(* IEC 61131-3 sources: Yaha/Documentation/Infomaterial/OSCAT/pcworx_basic_333/module_export (part 3) *)

(* ---- DT_TO_STRF.ST ---- *)
(*@PROPERTIES_EX@
TYPE: POU
LOCALE: 0
IEC_LANGUAGE: ST
PLC_TYPE: independent
PROC_TYPE: independent
GROUP: STRINGS
*)
(*@KEY@:DESCRIPTION*)
version 1.1	19. oct. 2008
programmer 	hugo
tested by	oscat

DT_TO_STRINGF converts a DATETIME input to a formatted string
(*@KEY@:END_DESCRIPTION*)
FUNCTION_BLOCK DT_TO_STRF

(*Group:NewGroup*)

VAR_INPUT
	DTI :	UDINT;
	MS :	INT;
	FMT :	STRING;
	LANG :	INT;
END_VAR

VAR_OUTPUT
	DT_TO_STRF :	STRING;
END_VAR

VAR
	FILL :	oscat_STRING1 := STRING#'0';
	BLANK :	oscat_STRING1 := STRING#' ';
	ly :	INT;
	dx :	UDINT;
	fs :	oscat_STRING10;
	fs_tmp :	oscat_STRING10;
	td :	UDINT;
	tmp :	INT;
	pos :	INT;
	f :	INT;
	CODE :	CODE;
	MONTH_TO_STRING :	MONTH_TO_STRING;
	WEEKDAY_TO_STRING :	WEEKDAY_TO_STRING;
END_VAR

(*@KEY@: WORKSHEET
NAME: DT_TO_STRF
IEC_LANGUAGE: ST
*)
IF LANG < 1 THEN ly := 1; ELSE ly := MIN(2, LANG); END_IF;

(* decode date and time information *)
dx := DT_TO_DATE(DTI);
td := DT_TO_TOD(DTI);

(* parse the format string *)
DT_TO_STRF := FMT;
pos := FIND(DT_TO_STRF, '#');
WHILE pos > 0 DO
	(* retrieve format identifier *)
    CODE(STR:=DT_TO_STRF,POS:=pos + 1);
    f := _BYTE_TO_INT(CODE.CODE);
	(* generate the return string according to the format character *)
	fs := '';
	CASE f OF
         0: RETURN; (* illegal character index *)

		65 : (* letter A retunrs the year in 4 digits *)
			fs := INT_TO_STRING(YEAR_OF_DATE(dx),'%d');
		66 : (* letter B returns the year in exactly 2 digits *)
			fs := RIGHT(INT_TO_STRING(YEAR_OF_DATE(dx),'%02d'),2);
		67 : (* letter C returns the month with 1 or 2 digits *)
			fs := INT_TO_STRING(MONTH_OF_DATE(dx),'%d');
		68 : (* letter D returns the month with exactly 2 digits *)
			fs := INT_TO_STRING(MONTH_OF_DATE(dx),'%02d');
		69 : (* letter E returns the month with 3 characters *)
            MONTH_TO_STRING(MTH:=MONTH_OF_DATE(dx),LANG:=ly,LX:=3);
            fs:=MONTH_TO_STRING.MONTH_TO_STRING;
		70 : (* letter F returns the month with all characters *)
            MONTH_TO_STRING(MTH:=MONTH_OF_DATE(dx),LANG:=ly,LX:=0);
            fs:=MONTH_TO_STRING.MONTH_TO_STRING;
		71 : (* letter G returns the day with up to 2 digits *)
			fs := INT_TO_STRING(DAY_OF_MONTH(dx),'%d');
		72 : (* letter H returns the day of the month with exactly 2 digits *)
			fs := INT_TO_STRING(DAY_OF_MONTH(dx),'%d');
			IF LEN(fs) < 2 THEN fs_tmp:=fs; fs := CONCAT(FILL, fs_tmp); END_IF;
		73 : (* letter I returns the weekday as the number 1..7 1 = monday *)
			fs := INT_TO_STRING(DAY_OF_WEEK(dx),'%d');
		74 : (* letter J returns the weekday in 2 character writing *)
            WEEKDAY_TO_STRING(WDAY:=DAY_OF_WEEK(dx),LANG:=ly,LX:=2);
            fs := WEEKDAY_TO_STRING.WEEKDAY_TO_STRING;
		75 : (* letter K returns the weekday with all characters *)
            WEEKDAY_TO_STRING(WDAY:=DAY_OF_WEEK(dx),LANG:=ly,LX:=0);
            fs := WEEKDAY_TO_STRING.WEEKDAY_TO_STRING;
		76 : (* letter L returns AM or PM for the given DateTime *)
			IF td >= UDINT#43200000 THEN fs := 'PM'; ELSE fs := 'AM'; END_IF;
		77 : (* letter M returns the hour in 1 or 2 digit form 0..24h *)
			fs := INT_TO_STRING(HOUR(td),'%d');
		78 : (* letter N returns the hour in exactly 2 digit form 0..24h *)
			fs := INT_TO_STRING(HOUR(td),'%d');
			IF LEN(fs) < 2 THEN fs_tmp:=fs; fs := CONCAT(FILL, fs_tmp); END_IF;
		79 : (* letter O returns the hour in 1 or 2 digit form 0..12h *)
			tmp := HOUR(td) MOD 12;
			IF tmp = 0 THEN tmp := 12; END_IF;
			fs := INT_TO_STRING(tmp,'%d');
		80 : (* letter P returns the hour in exactly 2 digit form 0..12h *)
			tmp := HOUR(td) MOD 12;
			IF tmp = 0 THEN tmp := 12; END_IF;
			fs := INT_TO_STRING(tmp,'%d');
			IF LEN(fs) < 2 THEN fs_tmp:=fs; fs := CONCAT(FILL, fs_tmp); END_IF;
		81 : (* letter Q returns the minute of the hour in 1 or two digit form *)
			fs := INT_TO_STRING(MINUTE(td),'%d');
		82 : (* letter R returns the minute of the hour in exactly two digit form *)
			fs := INT_TO_STRING(MINUTE(td),'%d');
			IF LEN(fs) < 2 THEN fs_tmp:=fs; fs := CONCAT(FILL, fs_tmp); END_IF;
		83 : (* letter S returns the second of the minute in 1 or two digit form *)
			fs := INT_TO_STRING(REAL_TO_INT(SECOND(td)),'%d');
		84 : (* letter T returns the second of the minute in exactly two digit form *)
			fs := INT_TO_STRING(REAL_TO_INT(SECOND(td)),'%d');
			IF LEN(fs) < 2 THEN fs_tmp:=fs; fs := CONCAT(FILL, fs_tmp); END_IF;
		85 : (* letter U returns the milliseconds in 1 to 3 digits *)
			fs := INT_TO_STRING(MS,'%d');
		86 : (* letter V returns the milliseconds in exactly 3 digit form *)
			fs := INT_TO_STRING(MS,'%03d');
		87 : (* letter W returns the day of the month with exactly 2 digits first digit is filled with blank if necessary *)
			fs := INT_TO_STRING(DAY_OF_MONTH(dx),'%d');
			IF LEN(fs) < 2 THEN fs_tmp:=fs; fs := CONCAT(BLANK, fs_tmp); END_IF;
		88 : (* letter X returns the month with exactly 2 digits first digit is filled with blank if necessary *)
			fs := INT_TO_STRING(MONTH_OF_DATE(dx),'%d');
			IF LEN(fs) < 2 THEN fs_tmp:=fs; fs := CONCAT(BLANK, fs_tmp); END_IF;
	END_CASE;
	DT_TO_STRF := REPLACE(DT_TO_STRF, fs, 2, pos);
	pos := FIND(DT_TO_STRF, '#');
END_WHILE;

(* revision history
hm	7. oct. 2008	rev 1.0
	original version

hm	19. oct. 2008	rev 1.1
	changed language setup constants
*)
(*@KEY@: END_WORKSHEET *)
END_FUNCTION_BLOCK

(* ---- DT_TO_STRING.ST ---- *)
(*@PROPERTIES_EX@
TYPE: POU
LOCALE: 0
IEC_LANGUAGE: ST
PLC_TYPE: independent
PROC_TYPE: independent
GROUP: EMULATION
*)
(*@KEY@:DESCRIPTION*)

(*@KEY@:END_DESCRIPTION*)
FUNCTION_BLOCK DT_TO_STRING

(*Group:Default*)

VAR_INPUT
	IDT :	UDINT;
END_VAR

VAR_OUTPUT
	DT_STRING :	STRING;
END_VAR

VAR
	st_tmp1 :	STRING;
	st_tmp2 :	STRING;
END_VAR

(*@KEY@: WORKSHEET
NAME: DT_TO_STRING
IEC_LANGUAGE: ST
*)
st_tmp2 := CONCAT(INT_TO_STRING(YEAR_OF_DATE(IDT),'%04d-'),INT_TO_STRING(MONTH_OF_DATE(IDT),'%02d-'));
st_tmp1 := CONCAT(INT_TO_STRING(day_of_month(IDT),'%02d-'),INT_TO_STRING(hour_of_DT(IDT),'%02d:'));
st_tmp2 := CONCAT(st_tmp2,st_tmp1);
st_tmp1 := CONCAT(INT_TO_STRING(minute_of_DT(IDT),'%02d:'),INT_TO_STRING(second_of_DT(IDT),'%02d'));
st_tmp2 := CONCAT(st_tmp2,st_tmp1);
DT_STRING := st_tmp2;
(*@KEY@: END_WORKSHEET *)
END_FUNCTION_BLOCK

(* ---- DW_TO_REAL.ST ---- *)
(*@PROPERTIES_EX@
TYPE: POU
LOCALE: 0
IEC_LANGUAGE: ST
PLC_TYPE: independent
PROC_TYPE: independent
GROUP: LOGIC.GATE_LOGIC
*)
(*@KEY@:DESCRIPTION*)
version 1.0	18. apr. 2008
programmer 	hugo
tested by	tobias

this function converts a DWORD to REAL in a bitwise manner.
(*@KEY@:END_DESCRIPTION*)
FUNCTION_BLOCK DW_TO_REAL

(*Group:Default*)

VAR_INPUT
	X :	DWORD;
END_VAR

VAR_OUTPUT
	DW_TO_REAL :	REAL;
END_VAR

VAR
	BUF_TO_REAL :	BUF_TO_REAL;
	i :	INT;
END_VAR

(*@KEY@: WORKSHEET
NAME: DW_TO_REAL
IEC_LANGUAGE: ST
*)
(* BUF_TO_REAL muss mit positiver Flanke gstartet werden darum wird dieser *)
(* einmal mit REQ=0 und dann mit REQ=1 aufgerufen                          *)
(* somit kann in jeden zyklus kopiert werden                               *)

FOR I := 0 TO 1 DO
  BUF_TO_REAL.REQ        := I > 0;
  BUF_TO_REAL.BUF_FORMAT := FALSE;
  BUF_TO_REAL.BUF_OFFS   := DINT#0;
  BUF_TO_REAL.BUF_CNT    := DINT#4;
  BUF_TO_REAL.BUFFER     := X;
  BUF_TO_REAL.DST        := DW_TO_REAL;
  BUF_TO_REAL();
  X           := BUF_TO_REAL.BUFFER;
  DW_TO_REAL  := BUF_TO_REAL.DST;
END_FOR;
(*@KEY@: END_WORKSHEET *)
END_FUNCTION_BLOCK

(* ---- DWORD_TO_STRB.ST ---- *)
(*@PROPERTIES_EX@
TYPE: POU
LOCALE: 0
IEC_LANGUAGE: ST
PLC_TYPE: independent
PROC_TYPE: independent
GROUP: STRINGS
*)
(*@KEY@:DESCRIPTION*)
version 1.3	20. jun. 2008
programmer 	hugo
tested by	oscat

DWORD_TO_STRINGB converts a DWORD to a String of Bits represented by '0' and '1' s.
The lowest order bit will be on the right and the high order bit on the left.
(*@KEY@:END_DESCRIPTION*)
FUNCTION_BLOCK DWORD_TO_STRB

(*Group:Default*)

VAR_INPUT
	IN :	DWORD;
END_VAR

VAR_OUTPUT
	DWORD_TO_STRB :	oscat_STRING32;
END_VAR

VAR
	i :	INT;
END_VAR

(*@KEY@: WORKSHEET
NAME: DWORD_TO_STRB
IEC_LANGUAGE: ST
*)
DWORD_TO_STRB :='';
FOR i := 1 TO 32 DO
    IF (in AND DWORD#16#8000_0000) > DWORD#0 THEN
        DWORD_TO_STRB := CONCAT(DWORD_TO_STRB,'1');
    ELSE
        DWORD_TO_STRB := CONCAT(DWORD_TO_STRB,'0');
    END_IF;
	in := SHL(in, 1);
END_FOR;

(* revision history
hm		9.6.2007	rev 1.0
	original version

hm		15.dec 2007	rev 1.1
	changed code for better performance

hm	29. mar. 2008	rev 1.2
	changed STRING to STRING(32)

hm	20. jun. 2008	rev 1.3
	performance improvement

*)
(*@KEY@: END_WORKSHEET *)
END_FUNCTION_BLOCK

(* ---- DWORD_TO_STRF.ST ---- *)
(*@PROPERTIES_EX@
TYPE: POU
LOCALE: 0
IEC_LANGUAGE: ST
PLC_TYPE: independent
PROC_TYPE: independent
GROUP: STRINGS
*)
(*@KEY@:DESCRIPTION*)
version 1.0	26 jan 2007
programmer 	hugo
tested by		tobias

dword_to_strF converts a DWORD, BYTE or Word to a fixed length String.
the string will be filled with leading zeroes to achieve the fixed length, or if too long, the lowest digits will be used.
the maximum allowed length is 20 mdigits.

for example:	dword_to_strf(123,4) = '0123'
				dword_to_strf(123,2) = '23'
(*@KEY@:END_DESCRIPTION*)
FUNCTION_BLOCK DWORD_TO_STRF

(*Group:Default*)

VAR_INPUT
	IN :	DWORD;
	N :	INT;
END_VAR

VAR_OUTPUT
	DWORD_TO_STRF :	STRING;
END_VAR

VAR
	FIX :	FIX;
END_VAR

(*@KEY@: WORKSHEET
NAME: DWORD_TO_STRF
IEC_LANGUAGE: ST
*)
(* limit N to max 20 characters *)
(* convert dword to string first and cut to length N *)
FIX(str:=DWORD_TO_STRING(in,'%u'),L:=LIMIT(0,N,20),C:=BYTE#48,M:=1);
DWORD_TO_STRF:=FIX.FIX;

(* old code

temp := DWORD_TO_STRING(in,STRING#'%u');
L := LEN(temp);
IF N < L THEN
    temp :=RIGHT(temp,N);
    L := N;
END_IF;

WHILE L < N DO
    temp2 := temp;
	temp := CONCAT('0', temp2);
	L := L + 1;
END_WHILE;
DWORD_TO_STRF := temp;

*)

(* revision history
hm	26. jan.2007	rev 1.0
	original version

hm	29. mar. 2008	rev 1.1
	changed STRING to STRING(20)
	limit the output string to max 20 digits
*)
(*@KEY@: END_WORKSHEET *)
END_FUNCTION_BLOCK

(* ---- DWORD_TO_STRH.ST ---- *)
(*@PROPERTIES_EX@
TYPE: POU
LOCALE: 0
IEC_LANGUAGE: ST
PLC_TYPE: independent
PROC_TYPE: independent
GROUP: STRINGS
*)
(*@KEY@:DESCRIPTION*)
version 1.3	29. mar. 2008
programmer 	hugo
tested by	tobias

DWORD_TO_STRINGH converts a DWORD to a String of Hexadecimal represented by '0' .. '9' and 'A' .. 'F'.
The lowest order Character will be on the right and the high order Character on the left.
(*@KEY@:END_DESCRIPTION*)
FUNCTION_BLOCK DWORD_TO_STRH

(*Group:Default*)

VAR_INPUT
	IN :	DWORD;
END_VAR

VAR_OUTPUT
	DWORD_TO_STRH :	STRING;
END_VAR

(*@KEY@: WORKSHEET
NAME: DWORD_TO_STRH
IEC_LANGUAGE: ST
*)
DWORD_TO_STRH:=DWORD_TO_STRING(IN,'%08X');

(* old code
temp :='';
FOR i := 1 TO 8 DO
	X := DWORD_TO_INT(in AND DWORD#2#1111);
	IF X <= 9 THEN X := X + 48; ELSE X := X + 55; END_IF;

    CHR(C:=INT_TO_BYTE(X));

    temp2 := temp;
	temp := CONCAT(CHR.CHR, temp2);
	in := SHR(in,4);
END_FOR;
DWORD_TO_STRH := temp;
*)

(* revision history
hm	9. jun. 2007	rev 1.0
	original version

hm	11. sep. 2007	rev 1.1
	changed coding for compatibility with twincat, concat cannot support a function as an argument.

hm	15. dec. 2007	rev 1.2
	changed code for better performance

hm	29. mar. 2008	rev 1.3
	changed STRING to STRING(8)

*)
(*@KEY@: END_WORKSHEET *)
END_FUNCTION_BLOCK

(* ---- ENERGY.ST ---- *)
(*@PROPERTIES_EX@
TYPE: POU
LOCALE: 0
IEC_LANGUAGE: ST
PLC_TYPE: independent
PROC_TYPE: independent
GROUP: ENGINEERING.CONVERSION
*)
(*@KEY@:DESCRIPTION*)
version 1.2	16. jan. 2010
programmer 	hugo
tested by	oscat

this function converts different energy units
any unused input can simply be left open.
different inputs connected at the same time will be added up.
(*@KEY@:END_DESCRIPTION*)
FUNCTION_BLOCK ENERGY

(*Group:Default*)

VAR_INPUT
	J :	REAL;
	C :	REAL;
	WH :	REAL;
END_VAR

VAR_OUTPUT
	YJ :	REAL;
	YC :	REAL;
	YWH :	REAL;
END_VAR

(*@KEY@: WORKSHEET
NAME: ENERGY
IEC_LANGUAGE: ST
*)
YJ := J + Wh * 3600.0 + C * 4.1868;
YC := YJ * 0.238845896627496;
YWh := YJ * 2.7777777778E-004;

(*
Arbeit, Energie, Joule* J 1 J = 1 N · m = 1 W · s = (1/3,6) E–6 kW · h = 1 kg · m2/s2
Wärmemenge Kilowattstunde kW · h 1 kW · h = 3,6 MJ = 860 kcal
Elektronvolt eV 1 eV = 160,218 92 E–21 J
Erg erg 1 erg = 1E–7 J
Kalorie calorie 1 calalorie = 4,1868 J = 1,163 E–3 W · h
Therm therm 1 therm = 105,50 · 106 J
*)

(* revision history

hm	27. mar. 2007	rev 1.0
	original version

hm	11. mar. 2009	rev 1.1
	improved code

hm 16. jan 2010	rev 1.2
	avoid the string cal in comments for codesys import bug

*)
(*@KEY@: END_WORKSHEET *)
END_FUNCTION_BLOCK

(* ---- ESR_COLLECT.ST ---- *)
(*@PROPERTIES_EX@
TYPE: POU
LOCALE: 0
IEC_LANGUAGE: ST
PLC_TYPE: independent
PROC_TYPE: independent
GROUP: OTHER
*)
(*@KEY@:DESCRIPTION*)
version 1.4	1. dec. 2009
programmer 	hugo
tested by	tobias

ESR_collect collects esr data from up to 8 esr_mon modules and stroes them in an output array.
the output pos will display the position of the last element in the array. if the array is empty, pos = -1
when to buffer is read by followon modules. pos has to be reset to -1
if the array will be full, the buffer will be refilled starting at position 0.

(*@KEY@:END_DESCRIPTION*)
FUNCTION_BLOCK ESR_COLLECT

(*Group:Default*)

VAR_INPUT
	ESR_0 :	oscat_ESR_3;
	ESR_1 :	oscat_ESR_3;
	ESR_2 :	oscat_ESR_3;
	ESR_3 :	oscat_ESR_3;
	ESR_4 :	oscat_ESR_3;
	ESR_5 :	oscat_ESR_3;
	ESR_6 :	oscat_ESR_3;
	ESR_7 :	oscat_ESR_3;
	RST :	BOOL;
END_VAR

VAR_IN_OUT
	POS :	INT;
END_VAR

VAR_OUTPUT
	ESR_OUT :	oscat_ESR_31;
END_VAR

VAR
	cnt :	INT := -1;
	max_in :	INT := 3;
	max_out :	INT := 32;
END_VAR

(*@KEY@: WORKSHEET
NAME: ESR_COLLECT
IEC_LANGUAGE: ST
*)
IF rst OR cnt < 0 THEN
	pos := -1;
ELSE
	FOR cnt := 0 TO max_in DO
	IF esr_0[cnt].typ > BYTE#0 THEN pos := INC1(pos, max_out); esr_out[pos] := esr_0[cnt]; END_IF;
	IF esr_1[cnt].typ > BYTE#0 THEN pos := INC1(pos, max_out); esr_out[pos] := esr_1[cnt]; END_IF;
	IF esr_2[cnt].typ > BYTE#0 THEN pos := INC1(pos, max_out); esr_out[pos] := esr_2[cnt]; END_IF;
	IF esr_3[cnt].typ > BYTE#0 THEN pos := INC1(pos, max_out); esr_out[pos] := esr_3[cnt]; END_IF;
	IF esr_4[cnt].typ > BYTE#0 THEN pos := INC1(pos, max_out); esr_out[pos] := esr_4[cnt]; END_IF;
	IF esr_5[cnt].typ > BYTE#0 THEN pos := INC1(pos, max_out); esr_out[pos] := esr_5[cnt]; END_IF;
	IF esr_6[cnt].typ > BYTE#0 THEN pos := INC1(pos, max_out); esr_out[pos] := esr_6[cnt]; END_IF;
	IF esr_7[cnt].typ > BYTE#0 THEN pos := INC1(pos, max_out); esr_out[pos] := esr_7[cnt]; END_IF;
   END_FOR;
END_IF;

(* revision history
hm	26.jan 2007	rev 1.0
	original version

hm	8. dec 2007	rev 1.1
	added reset input

ks	27. oct. 2008	rev 1.2
	optimized code for performance

ks	12. nov. 2009	rev 1.3
	output pos was not pointing to last value

hm	1. dec. 2009	rev 1.4
	changed pos to be I/O
	reduced output array size to 32 elements
*)
(*@KEY@: END_WORKSHEET *)
END_FUNCTION_BLOCK

(* ---- ESR_MON_B8.ST ---- *)
(*@PROPERTIES_EX@
TYPE: POU
LOCALE: 0
IEC_LANGUAGE: ST
PLC_TYPE: independent
PROC_TYPE: independent
GROUP: OTHER
*)
(*@KEY@:DESCRIPTION*)
version 1.3	1. dec. 2009
programmer 	hugo
tested by	tobias

ESR_mon_B8 monitores up to 8 binary inputs and reports changes with time stamd and adress label.
the module checks 8 inputs for a change and reports all changes with time and adress stamp to the output.
4 events maximum can be collected at once within the same cycle

(*@KEY@:END_DESCRIPTION*)
FUNCTION_BLOCK ESR_MON_B8

(*Group:Default*)

VAR_INPUT
	S0 :	BOOL;
	A0 :	oscat_STRING10;
	S1 :	BOOL;
	A1 :	oscat_STRING10;
	S2 :	BOOL;
	A2 :	oscat_STRING10;
	S3 :	BOOL;
	A3 :	oscat_STRING10;
	S4 :	BOOL;
	A4 :	oscat_STRING10;
	S5 :	BOOL;
	A5 :	oscat_STRING10;
	S6 :	BOOL;
	A6 :	oscat_STRING10;
	S7 :	BOOL;
	A7 :	oscat_STRING10;
	DT_IN :	UDINT;
END_VAR

VAR_IN_OUT
	ESR_Out :	oscat_ESR_3;
END_VAR

VAR_OUTPUT
	ESR_FLAG :	BOOL;
END_VAR

VAR
	x0 :	BOOL;
	x1 :	BOOL;
	x2 :	BOOL;
	x3 :	BOOL;
	x4 :	BOOL;
	x5 :	BOOL;
	x6 :	BOOL;
	x7 :	BOOL;
	tx :	TIME;
	cnt :	INT;
	T_PLC_MS :	T_PLC_MS;
END_VAR

(*@KEY@: WORKSHEET
NAME: ESR_MON_B8
IEC_LANGUAGE: ST
*)
(* read system timer *)
T_PLC_MS();
tx:= UDINT_TO_TIME(T_PLC_MS.T_PLC_MS);

ESR_Flag := FALSE;
esr_out[3].typ := BYTE#0;
esr_out[2].typ := BYTE#0;
esr_out[1].typ := BYTE#0;
esr_out[0].typ := BYTE#0;
cnt := 0;

(* check if inputs have chaged and fill buffer *)
IF s0 <> X0 THEN
	esr_out[cnt].typ := INT_TO_BYTE(10 + BOOL_TO_INT(s0));
	esr_out[cnt].adress := a0;
	esr_out[cnt].DS := DT_in;
	esr_out[cnt].TS := TX;
	X0 := S0;
	cnt := cnt + 1;
	esr_flag := TRUE;
END_IF;
IF s1 <> X1 THEN
	esr_out[cnt].typ := INT_TO_BYTE(10 + BOOL_TO_INT(s1));
	esr_out[cnt].adress := a1;
	esr_out[cnt].DS := DT_in;
	esr_out[cnt].TS := TX;
	X1 := S1;
	cnt := cnt + 1;
	esr_flag := TRUE;
END_IF;
IF s2 <> X2 THEN
	esr_out[cnt].typ := INT_TO_BYTE(10 + BOOL_TO_INT(s2));
	esr_out[cnt].adress := a2;
	esr_out[cnt].DS := DT_in;
	esr_out[cnt].TS := TX;
	X2 := S2;
	cnt := cnt + 1;
	esr_flag := TRUE;
END_IF;
IF s3 <> X3 THEN
	esr_out[cnt].typ := INT_TO_BYTE(10 + BOOL_TO_INT(s3));
	esr_out[cnt].adress := a3;
	esr_out[cnt].DS := DT_in;
	esr_out[cnt].TS := TX;
	X3 := S3;
	cnt := cnt + 1;
	esr_flag := TRUE;
END_IF;
IF s4 <> X4 AND cnt < 4 THEN
	esr_out[cnt].typ := INT_TO_BYTE(10 + BOOL_TO_INT(s4));
	esr_out[cnt].adress := a4;
	esr_out[cnt].DS := DT_in;
	esr_out[cnt].TS := TX;
	X4 := S4;
	cnt := cnt + 1;
	esr_flag := TRUE;
END_IF;
IF s5 <> X5  AND cnt < 4 THEN
	esr_out[cnt].typ := INT_TO_BYTE(10 + BOOL_TO_INT(s5));
	esr_out[cnt].adress := a5;
	esr_out[cnt].DS := DT_in;
	esr_out[cnt].TS := TX;
	X5 := S5;
	cnt := cnt + 1;
	esr_flag := TRUE;
END_IF;
IF s6 <> X6  AND cnt < 4 THEN
	esr_out[cnt].typ := INT_TO_BYTE(10 + BOOL_TO_INT(s6));
	esr_out[cnt].adress := a6;
	esr_out[cnt].DS := DT_in;
	esr_out[cnt].TS := TX;
	X6 := S6;
	cnt := cnt + 1;
	esr_flag := TRUE;
END_IF;
IF s7 <> X7  AND cnt < 4 THEN
	esr_out[cnt].typ := INT_TO_BYTE(10 + BOOL_TO_INT(s7));
	esr_out[cnt].adress := a7;
	esr_out[cnt].DS := DT_in;
	esr_out[cnt].TS := TX;
	X7 := S7;
	cnt := cnt + 1;
	esr_flag := TRUE;
END_IF;

(* revision history
hm	26. jan 2007	rev 1.0
	original version

hm	17. sep 2007	rev 1.1
	replaced time() with T_PLC_MS() for compatibility reasons

hm	22. oct. 2008	rev 1.2
	optimized code

hm	1.dec. 2009	rev 1.3
	changed esr_out to be I/O

*)
(*@KEY@: END_WORKSHEET *)
END_FUNCTION_BLOCK

(* ---- ESR_MON_R4.ST ---- *)
(*@PROPERTIES_EX@
TYPE: POU
LOCALE: 0
IEC_LANGUAGE: ST
PLC_TYPE: independent
PROC_TYPE: independent
GROUP: OTHER
*)
(*@KEY@:DESCRIPTION*)
version 1.4	1. dec. 2009
programmer 	hugo
tested by	tobias

ESR_mon_R4 monitores up to 4 Real inputs and reports changes with time stamd and adress label.
the module checks 4 inputs for a change of more than the specified sensitivity S and reports all changes with time and adress stamp to the output.

(*@KEY@:END_DESCRIPTION*)
FUNCTION_BLOCK ESR_MON_R4

(*Group:Default*)

VAR_INPUT
	R0 :	REAL;
	A0 :	oscat_STRING10;
	S0 :	REAL;
	R1 :	REAL;
	A1 :	oscat_STRING10;
	S1 :	REAL;
	R2 :	REAL;
	A2 :	oscat_STRING10;
	S2 :	REAL;
	R3 :	REAL;
	A3 :	oscat_STRING10;
	S3 :	REAL;
	DT_IN :	UDINT;
END_VAR

VAR_IN_OUT
	ESR_OUT :	oscat_ESR_3;
END_VAR

VAR_OUTPUT
	ESR_FLAG :	BOOL;
END_VAR

VAR
	x0 :	REAL;
	x1 :	REAL;
	x2 :	REAL;
	x3 :	REAL;
	tx :	TIME;
	cnt :	INT;
	T_PLC_MS :	T_PLC_MS;
	REAL_TO_DW :	REAL_TO_DW;
	tmp :	DWORD;
END_VAR

(*@KEY@: WORKSHEET
NAME: ESR_MON_R4
IEC_LANGUAGE: ST
*)
T_PLC_MS();
tx:= UDINT_TO_TIME(T_PLC_MS.T_PLC_MS);

ESR_Flag := FALSE;
esr_out[3].typ := BYTE#0;
esr_out[2].typ := BYTE#0;
esr_out[1].typ := BYTE#0;
esr_out[0].typ := BYTE#0;
cnt := 0;

(* check if inputs have chaged and fill buffer *)
IF differ(R0, X0, S0) THEN
    REAL_TO_DW(X:=R0);
    tmp := REAL_TO_DW.REAL_TO_DW;

	esr_out[cnt].typ := BYTE#20;
	esr_out[cnt].adress := a0;
	esr_out[cnt].DS := DT_in;
	esr_out[cnt].TS := TX;
	esr_out[cnt].data[0] := Byte_of_Dword(tmp,BYTE#0);
	esr_out[cnt].data[1] := Byte_of_Dword(tmp,BYTE#1);
	esr_out[cnt].data[2] := Byte_of_Dword(tmp,BYTE#2);
	esr_out[cnt].data[3] := Byte_of_Dword(tmp,BYTE#3);
	X0 := R0;
	cnt := cnt + 1;
	esr_flag := TRUE;
END_IF;
IF differ(R1, X1, S1) THEN
    REAL_TO_DW(X:=R1);
    tmp := REAL_TO_DW.REAL_TO_DW;

	esr_out[cnt].typ := BYTE#20;
	esr_out[cnt].adress := a1;
	esr_out[cnt].DS := DT_in;
	esr_out[cnt].TS := TX;
	esr_out[cnt].data[0] := Byte_of_Dword(tmp,BYTE#0);
	esr_out[cnt].data[1] := Byte_of_Dword(tmp,BYTE#1);
	esr_out[cnt].data[2] := Byte_of_Dword(tmp,BYTE#2);
	esr_out[cnt].data[3] := Byte_of_Dword(tmp,BYTE#3);
	X1 := R1;
	cnt := cnt + 1;
	esr_flag := TRUE;
END_IF;
IF differ(R2, X2, S2) THEN
    REAL_TO_DW(X:=R2);
    tmp := REAL_TO_DW.REAL_TO_DW;

	esr_out[cnt].typ := BYTE#20;
	esr_out[cnt].adress := a2;
	esr_out[cnt].DS := DT_in;
	esr_out[cnt].TS := TX;
	esr_out[cnt].data[0] := Byte_of_Dword(tmp,BYTE#0);
	esr_out[cnt].data[1] := Byte_of_Dword(tmp,BYTE#1);
	esr_out[cnt].data[2] := Byte_of_Dword(tmp,BYTE#2);
	esr_out[cnt].data[3] := Byte_of_Dword(tmp,BYTE#3);
	X2 := R2;
	cnt := cnt + 1;
	esr_flag := TRUE;
END_IF;
IF differ(R3, X3, S3) THEN
    REAL_TO_DW(X:=R2);
    tmp := REAL_TO_DW.REAL_TO_DW;

	esr_out[cnt].typ := BYTE#20;
	esr_out[cnt].adress := a3;
	esr_out[cnt].DS := DT_in;
	esr_out[cnt].TS := TX;
	esr_out[cnt].data[0] := Byte_of_Dword(tmp,BYTE#0);
	esr_out[cnt].data[1] := Byte_of_Dword(tmp,BYTE#1);
	esr_out[cnt].data[2] := Byte_of_Dword(tmp,BYTE#2);
	esr_out[cnt].data[3] := Byte_of_Dword(tmp,BYTE#3);
	X3 := R3;
	cnt := cnt + 1;
	esr_flag := TRUE;
END_IF;

(* revision history
hm	26. jan 2007	rev 1.0
	original version

hm	17. sep. 2007		rev 1.1
	replaced time() with T_PLC_MS() for compatibility reasons

hm	8. dec. 2007		rev 1.2
	corrected an error while esr typ would not be set

hm	16. mar. 2008		rev 1.3
	deleted wrong conversion real_to_dword

hm	1. dec 2009		rev 1.4
	changed esr_out to be I/O

*)

(*@KEY@: END_WORKSHEET *)
END_FUNCTION_BLOCK

(* ---- ESR_MON_X8.ST ---- *)
(*@PROPERTIES_EX@
TYPE: POU
LOCALE: 0
IEC_LANGUAGE: ST
PLC_TYPE: independent
PROC_TYPE: independent
GROUP: OTHER
*)
(*@KEY@:DESCRIPTION*)
version 1.2	1. dec. 2009
programmer 	hugo
tested by	tobias

ESR_MON_X8 is a status and error collector.
the module checks 8 status inputs for a change and reports up to 4 input changes with time and adress stamp to the output.
the mode can be
1 for error only
2 for error and status
3 for error, status and debug
the adress label of the 8 inputs can be configured individually.
(*@KEY@:END_DESCRIPTION*)
FUNCTION_BLOCK ESR_MON_X8

(*Group:Default*)

VAR_INPUT
	S0 :	BYTE;
	A0 :	oscat_STRING10;
	S1 :	BYTE;
	A1 :	oscat_STRING10;
	S2 :	BYTE;
	A2 :	oscat_STRING10;
	S3 :	BYTE;
	A3 :	oscat_STRING10;
	S4 :	BYTE;
	A4 :	oscat_STRING10;
	S5 :	BYTE;
	A5 :	oscat_STRING10;
	S6 :	BYTE;
	A6 :	oscat_STRING10;
	S7 :	BYTE;
	A7 :	oscat_STRING10;
	DT_IN :	UDINT;
	MODE :	BYTE := BYTE#3;
END_VAR

VAR_IN_OUT
	ESR_OUT :	oscat_ESR_3;
END_VAR

VAR_OUTPUT
	ESR_FLAG :	BOOL;
END_VAR

VAR
	x0 :	BYTE;
	x1 :	BYTE;
	x2 :	BYTE;
	x3 :	BYTE;
	x4 :	BYTE;
	x5 :	BYTE;
	x6 :	BYTE;
	x7 :	BYTE;
	tx :	TIME;
	cnt :	INT;
	status_to_ESR :	status_to_ESR;
	T_PLC_MS :	T_PLC_MS;
END_VAR

(*@KEY@: WORKSHEET
NAME: ESR_MON_X8
IEC_LANGUAGE: ST
*)
(* read system timer *)
T_PLC_MS();
tx:= UDINT_TO_TIME(T_PLC_MS.T_PLC_MS);

ESR_Flag := FALSE;
esr_out[3].typ := BYTE#0;
esr_out[2].typ := BYTE#0;
esr_out[1].typ := BYTE#0;
esr_out[0].typ := BYTE#0;
cnt := 0;

(* check if inputs have chaged and fill buffer *)
IF s0 <> X0 AND ((s0 < BYTE#100) OR (S0 > BYTE#99 AND S0 < BYTE#200 AND mode >= BYTE#2) OR (S0 > BYTE#199 AND mode = BYTE#3)) THEN

    status_to_ESR.status := s0;
    status_to_ESR.adress := a0;
    status_to_ESR.DT_in  := DT_in;
    status_to_ESR.TS     := tx;
    status_to_ESR();
    esr_out[cnt] := status_to_ESR.status_to_ESR;

	X0 := S0;
	cnt := cnt + 1;
	esr_flag := TRUE;
END_IF;
IF s1 <> X1 AND ((s1 < BYTE#100) OR (S1 > BYTE#99 AND S1 < BYTE#200 AND mode >= BYTE#2) OR (S1 > BYTE#199 AND mode = BYTE#3)) THEN

    status_to_ESR.status := s1;
    status_to_ESR.adress := a1;
    status_to_ESR.DT_in  := DT_in;
    status_to_ESR.TS     := tx;
    status_to_ESR();
    esr_out[cnt] := status_to_ESR.status_to_ESR;

	X1 := S1;
	cnt := cnt + 1;
	esr_flag := TRUE;
END_IF;
IF s2 <> X2 AND ((s2 < BYTE#100) OR (S2 > BYTE#99 AND S2 < BYTE#200 AND mode >= BYTE#2) OR (S2 > BYTE#199 AND mode = BYTE#3)) THEN

    status_to_ESR.status := s2;
    status_to_ESR.adress := a2;
    status_to_ESR.DT_in  := DT_in;
    status_to_ESR.TS     := tx;
    status_to_ESR();
    esr_out[cnt] := status_to_ESR.status_to_ESR;

	X2 := S2;
	cnt := cnt + 1;
	esr_flag := TRUE;
END_IF;
IF s3 <> X3 AND ((s3 < BYTE#100) OR (S3 > BYTE#99 AND S3 < BYTE#200 AND mode >= BYTE#2) OR (S3 > BYTE#199 AND mode = BYTE#3)) THEN

    status_to_ESR.status := s3;
    status_to_ESR.adress := a3;
    status_to_ESR.DT_in  := DT_in;
    status_to_ESR.TS     := tx;
    status_to_ESR();
    esr_out[cnt] := status_to_ESR.status_to_ESR;

	X3 := S3;
	cnt := cnt + 1;
	esr_flag := TRUE;
END_IF;
IF cnt < 4 AND s4 <> X4 AND ((s4 < BYTE#100) OR (S4 > BYTE#99 AND S4 < BYTE#200 AND mode >= BYTE#2) OR (S4 > BYTE#199 AND mode = BYTE#3)) THEN

    status_to_ESR.status := s4;
    status_to_ESR.adress := a4;
    status_to_ESR.DT_in  := DT_in;
    status_to_ESR.TS     := tx;
    status_to_ESR();
    esr_out[cnt] := status_to_ESR.status_to_ESR;

	X4 := S4;
	cnt := cnt + 1;
	esr_flag := TRUE;
END_IF;
IF cnt < 4 AND s5 <> X5 AND ((s5 < BYTE#100) OR (S5 > BYTE#99 AND S5 < BYTE#200 AND mode >= BYTE#2) OR (S5 > BYTE#199 AND mode = BYTE#3)) THEN

    status_to_ESR.status := s5;
    status_to_ESR.adress := a5;
    status_to_ESR.DT_in  := DT_in;
    status_to_ESR.TS     := tx;
    status_to_ESR();
    esr_out[cnt] := status_to_ESR.status_to_ESR;

	X5 := S5;
	cnt := cnt + 1;
	esr_flag := TRUE;
END_IF;
IF cnt < 4 AND s6 <> X6 AND ((s6 < BYTE#100) OR (S6 > BYTE#99 AND S6 < BYTE#200 AND mode >= BYTE#2) OR (S6 > BYTE#199 AND mode = BYTE#3)) THEN

    status_to_ESR.status := s6;
    status_to_ESR.adress := a6;
    status_to_ESR.DT_in  := DT_in;
    status_to_ESR.TS     := tx;
    status_to_ESR();
    esr_out[cnt] := status_to_ESR.status_to_ESR;

	X6 := S6;
	cnt := cnt + 1;
	esr_flag := TRUE;
END_IF;
IF cnt < 4 AND s7 <> X7 AND ((s7 < BYTE#100) OR (S7 > BYTE#99 AND S7 < BYTE#200 AND mode >= BYTE#2) OR (S7 > BYTE#199 AND mode = BYTE#3)) THEN

    status_to_ESR.status := s7;
    status_to_ESR.adress := a7;
    status_to_ESR.DT_in  := DT_in;
    status_to_ESR.TS     := tx;
    status_to_ESR();
    esr_out[cnt] := status_to_ESR.status_to_ESR;

	X7 := S7;
	cnt := cnt + 1;
	esr_flag := TRUE;
END_IF;

(* revision history
hm	26. jan 2007		rev 1.0
	original version

hm	17. sep 2007	rev 1.1
	replaced time() with T_PLC_MS() for compatibility reasons

hm	1. dec. 2009	rev 1.2
	changed esr_out to be I/O

*)
(*@KEY@: END_WORKSHEET *)
END_FUNCTION_BLOCK

(* ---- EVENTS.ST ---- *)
(*@PROPERTIES_EX@
TYPE: POU
LOCALE: 0
IEC_LANGUAGE: ST
PLC_TYPE: independent
PROC_TYPE: independent
GROUP: TIME_DATE
*)
(*@KEY@:DESCRIPTION*)
version 1.0	18. jan. 2010
programmer 	hugo
tested by	tobias

event checks an array with a list of events and displays the event if today is one.

(*@KEY@:END_DESCRIPTION*)
FUNCTION_BLOCK EVENTS

(*Group:Default*)

VAR_INPUT
	DATE_IN :	UDINT;
	ENA :	BOOL;
END_VAR

VAR_OUTPUT
	Y :	BOOL;
	NAME :	oscat_STRING30;
END_VAR

VAR_IN_OUT
	ELIST :	oscat_HOLIDAY_DATA_0_49;
END_VAR

VAR
	i :	INT;
	last_active :	UDINT;
	size :	INT := 49;
	day_in :	DINT;
	cyr :	INT;
	lday :	DINT;
	check :	oscat_HOLIDAY_DATA;
	y_int :	BOOL;
	name_int :	oscat_STRING30;
END_VAR

(*@KEY@: WORKSHEET
NAME: EVENTS
IEC_LANGUAGE: ST
*)
(* for performance reasons only activate once a day *)
IF last_active <> date_in THEN
	last_active := DATE_IN;
	Y_int := FALSE;
	name_int := '';
	day_in := DAY_OF_DATE(DATE_IN);
	cyr := YEAR_OF_DATE(DATE_IN);

	(* search list for events *)
	FOR i := 0 TO size DO
		check := elist[i];
		lday := DAY_OF_DATE(SET_DATE(cyr,SINT_TO_INT(check.month), SINT_TO_INT(check.day)));
		IF day_in >= lday AND day_in <= lday + SINT_TO_DINT(check.use) - DINT#1 THEN
			y_int := TRUE;
			name_int := check.name;
			EXIT;
		END_IF;
	END_FOR;
END_IF;

IF ENA THEN
	Y := y_int;
	NAME := name_int;
ELSE
	Y := FALSE;
	NAME := '';
END_IF;

(* revision history
hm  18. jan. 2011	rev 1.0
	new module

*)

(*@KEY@: END_WORKSHEET *)
END_FUNCTION_BLOCK

(* ---- EXEC.ST ---- *)
(*@PROPERTIES_EX@
TYPE: POU
LOCALE: 0
IEC_LANGUAGE: ST
PLC_TYPE: independent
PROC_TYPE: independent
GROUP: STRINGS
*)
(*@KEY@:DESCRIPTION*)
version 1.4	29. mar. 2008
programmer 	hugo
tested by	tobias

exec executes a mathematical term and returns the result as a string
the term can only be a simple term without brackets and only one operator
allowed operastors are: (+, -, *, /, ^, sqrt, sin, cos, tan).
(*@KEY@:END_DESCRIPTION*)
FUNCTION_BLOCK EXEC

(*Group:Default*)

VAR_INPUT
	STR :	STRING;
END_VAR

VAR_OUTPUT
	EXEC :	STRING;
END_VAR

VAR
	pos :	INT;
	R1 :	REAL;
	R2 :	REAL;
	operator :	STRING;
	temp :	STRING;
	uppercase :	uppercase;
	trim :	trim;
	findB_num :	findB_num;
	findB_nonum :	findB_nonum;
END_VAR

(*@KEY@: WORKSHEET
NAME: EXEC
IEC_LANGUAGE: ST
*)
(* extract both numbers and operator *)

trim(str:=str);
temp:=trim.trim;

uppercase(str:=temp);
exec:=uppercase.uppercase;

findB_nonum(str:=exec);
pos :=findB_nonum.findB_nonum;

IF pos > 1 THEN
 temp := LEFT(EXEC,pos-1);
 findB_num(str:=temp);
 IF findB_num.findB_num > 0 THEN
   R1 := STRING_TO_REAL(temp);
 END_IF;
END_IF;
temp := RIGHT(exec,LEN(exec)-pos);
R2 := STRING_TO_REAL(temp);
exec := LEFT(exec,pos);

findB_num(str:=exec);
pos :=findB_num.findB_num;
operator := RIGHT(exec,LEN(exec) - pos);
IF EQ_STRING(operator,'') AND LEN(str) = 0 THEN
	exec := '';
	RETURN;
ELSIF EQ_STRING(operator,'') THEN
	exec := str;
	RETURN;
END_IF;
IF EQ_STRING(operator,'^') THEN
	exec := REAL_TO_STRING(EXPT(R1, R2),'%f');
ELSIF EQ_STRING(operator,'SQRT') THEN
	exec := REAL_TO_STRING(SQRT(R2),'%f');
ELSIF EQ_STRING(operator,'SIN') THEN
	exec := REAL_TO_STRING(SIN(r2),'%f');
ELSIF EQ_STRING(operator,'COS') THEN
	exec := REAL_TO_STRING(COS(r2),'%f');
ELSIF EQ_STRING(operator,'TAN') THEN
	exec := REAL_TO_STRING(TAN(R2),'%f');
ELSIF EQ_STRING(operator,'*') THEN
	exec := REAL_TO_STRING(R1 * R2,'%f');
ELSIF EQ_STRING(operator,'/') THEN
	IF R2 <> 0.0 THEN exec := REAL_TO_STRING(R1 / R2,'%f'); ELSE exec := 'ERROR'; END_IF;
ELSIF EQ_STRING(operator,'+') THEN
	exec := REAL_TO_STRING(r1 + r2,'%f');
ELSIF EQ_STRING(operator,'-') THEN
	exec := REAL_TO_STRING(r1 - r2,'%f');
ELSE
	exec := 'ERROR';
END_IF;
IF EQ_STRING(EXEC,'ERROR') THEN
	RETURN;
(* some systems deliver integer instead of real *)
ELSIF FIND(EXEC,'.') = 0 THEN
	EXEC := CONCAT(EXEC, '.0');
(* some systems deliver n. instead of n.0 ! *)
ELSE
 temp := RIGHT(EXEC,1);
 IF EQ_STRING(temp,'.') THEN
    EXEC := CONCAT(EXEC,'0');
  END_IF;
END_IF;

(* revision history

hm 	6.feb 2007		rev 1.1
	cos has to be written in uppercase
	divide by 0 will return an error

hm	5. mar. 2008	rev 1.2
	add a 0 to the string if a '.' is at the end of the string

hm	20. mar. 2008	rev 1.3
	make sure the function always returns a real value in the form of x.y

hm	29. mar. 2008	rev 1.4
	changed STRING to STRING(STRING_LENGTH)
*)
(*@KEY@: END_WORKSHEET *)
END_FUNCTION_BLOCK

(* ---- F_POLY.ST ---- *)
(*@PROPERTIES_EX@
TYPE: POU
LOCALE: 0
IEC_LANGUAGE: ST
PLC_TYPE: independent
PROC_TYPE: independent
GROUP: MATHEMATICAL.FUNCTIONS
*)
(*@KEY@:DESCRIPTION*)
version 1.1	18. mar. 2011
programmer 	hugo
tested by	tobias

this function calculates the polynom C[0] + C[1]*X^1 + C[2]*X^2 * C[3]*X^3 + C[4]*X^4 + C[5]*X^5 + C[6]*X^6 + C[7]*X^7

(*@KEY@:END_DESCRIPTION*)
FUNCTION_BLOCK F_POLY

(*Group:Default*)

VAR_INPUT
	X :	REAL;
	C :	oscat_arr_0_7;
END_VAR

VAR_OUTPUT
	F_POLY :	REAL;
END_VAR

(*@KEY@: WORKSHEET
NAME: F_POLY
IEC_LANGUAGE: ST
*)
F_POLY := ((((((( c[7] * x + c[6] ) * x + c[5] ) * x + c[4] ) * x + c[3] ) * x + c[2] ) * x + c[1] ) * x + c[0] ) ;

(* revision history
hm		20. may. 2008		rev 1.0
	original version

hm	18. mar. 2011	rev 1.1
	improved performance
*)

(*@KEY@: END_WORKSHEET *)
END_FUNCTION_BLOCK

(* ---- FADE.ST ---- *)
(*@PROPERTIES_EX@
TYPE: POU
LOCALE: 0
IEC_LANGUAGE: ST
PLC_TYPE: independent
PROC_TYPE: independent
GROUP: ENGINEERING.SIGNAL_PROCESSING
*)
(*@KEY@:DESCRIPTION*)
version 1.3	24. jan. 2009
programmer 	oscat
tested BY	oscat

FADE is used to crossfade between the inputs IN1 and IN2. The fade_over time is specified with TF.
When F = TRUE then Y = IN2 after the time TF, and when F = FALSE then Y = IN1.
(*@KEY@:END_DESCRIPTION*)
FUNCTION_BLOCK FADE

(*Group:Default*)

VAR_INPUT
	IN1 :	REAL;
	IN2 :	REAL;
	F :	BOOL;
	TF :	TIME;
	RST :	BOOL;
END_VAR

VAR_OUTPUT
	Y :	REAL;
END_VAR

VAR
	rmx :	RMP_W;
END_VAR

(*@KEY@: WORKSHEET
NAME: FADE
IEC_LANGUAGE: ST
*)
rmx(rst := rst AND NOT F, set := rst AND F, pt := TF, up := F);
Y := (in2 - In1) / 65535.0 * _WORD_TO_REAL(rmx.out) + in1;

(* revision history
hm	26. dec 2007	rev 1.0
	original version

hm	18. oct. 2008	rev 1.1
	improved performance
	changed calls for rmp_w because rmp_w has chaged

hm	17. dec. 2008	rev 1.2
	function of input f was inverted

hm	24. jan. 2009	rev 1.3
	delted unused var FF
*)
(*@KEY@: END_WORKSHEET *)
END_FUNCTION_BLOCK

(* ---- FF_D2E.ST ---- *)
(*@PROPERTIES_EX@
TYPE: POU
LOCALE: 0
IEC_LANGUAGE: ST
PLC_TYPE: independent
PROC_TYPE: independent
GROUP: LOGIC.FF_EDGE_TRIGGERED
*)
(*@KEY@:DESCRIPTION*)
version 1.3	14. mar. 2009
programmer 	hugo
tested by	oscat

dual D-type flip flop with reset and rising clock trigger
(*@KEY@:END_DESCRIPTION*)
FUNCTION_BLOCK FF_D2E

(*Group:Default*)

VAR_INPUT
	D0 :	BOOL;
	D1 :	BOOL;
	CLK :	BOOL;
	RST :	BOOL;
END_VAR

VAR_OUTPUT
	Q0 :	BOOL;
	Q1 :	BOOL;
END_VAR

VAR
	edge :	BOOL;
END_VAR

(*@KEY@: WORKSHEET
NAME: FF_D2E
IEC_LANGUAGE: ST
*)
IF rst THEN
	Q0 := FALSE;
	Q1 := FALSE;
ELSIF clk AND NOT edge THEN
	Q0 := D0;
	Q1 := D1;
END_IF;
edge := CLK;

(* revision history
hm	25. dec 2007	rev 1.0
	original version

hm	27. dec 2007	rev 1.1
	changed code for better performance

hm	30. oct. 200	rev 1.2
	deleted unnecessary init with 0

hm	14. mar. 2009	rev 1.3
	removed double assignments

*)

(*@KEY@: END_WORKSHEET *)
END_FUNCTION_BLOCK

(* ---- FF_D4E.ST ---- *)
(*@PROPERTIES_EX@
TYPE: POU
LOCALE: 0
IEC_LANGUAGE: ST
PLC_TYPE: independent
PROC_TYPE: independent
GROUP: LOGIC.FF_EDGE_TRIGGERED
*)
(*@KEY@:DESCRIPTION*)
version 1.3	14. mar. 2009
programmer 	hugo
tested by	oscat

quad D-type flip flop with reset and rising clock trigger

(*@KEY@:END_DESCRIPTION*)
FUNCTION_BLOCK FF_D4E

(*Group:Default*)

VAR_INPUT
	D0 :	BOOL;
	D1 :	BOOL;
	D2 :	BOOL;
	D3 :	BOOL;
	CLK :	BOOL;
	RST :	BOOL;
END_VAR

VAR_OUTPUT
	Q0 :	BOOL;
	Q1 :	BOOL;
	Q2 :	BOOL;
	Q3 :	BOOL;
END_VAR

VAR
	edge :	BOOL;
END_VAR

(*@KEY@: WORKSHEET
NAME: FF_D4E
IEC_LANGUAGE: ST
*)
IF rst THEN
	Q0 := FALSE;
	Q1 := FALSE;
	Q2 := FALSE;
	Q3 := FALSE;
ELSIF clk AND NOT edge THEN
	Q0 := D0;
	Q1 := D1;
	Q2 := D2;
	Q3 := D3;
END_IF;
edge := CLK;

(* revision history
hm	4. aug 2006	rev 1.0
	original version

hm	27. dec 2007	rev 1.1
	changed code for better performance

hm	30. oct. 200	rev 1.2
	deleted unnecessary init with 0

hm	14. mar. 2009	rev 1.3
	removed double assignments

*)

(*@KEY@: END_WORKSHEET *)
END_FUNCTION_BLOCK

(* ---- FF_DRE.ST ---- *)
(*@PROPERTIES_EX@
TYPE: POU
LOCALE: 0
IEC_LANGUAGE: ST
PLC_TYPE: independent
PROC_TYPE: independent
GROUP: LOGIC.FF_EDGE_TRIGGERED
*)
(*@KEY@:DESCRIPTION*)
version 1.2	30. oct. 2008
programmer 	hugo
tested by	oscat

D-type flip flop with set, reset and rising clock trigger
(*@KEY@:END_DESCRIPTION*)
FUNCTION_BLOCK FF_DRE

(*Group:Default*)

VAR_INPUT
	SET :	BOOL;
	D :	BOOL;
	CLK :	BOOL;
	RST :	BOOL;
END_VAR

VAR_OUTPUT
	Q :	BOOL;
END_VAR

VAR
	edge :	BOOL;
END_VAR

(*@KEY@: WORKSHEET
NAME: FF_DRE
IEC_LANGUAGE: ST
*)
IF rst OR set THEN
	Q := NOT rst;
ELSIF clk AND NOT edge THEN
	Q := D;
END_IF;
edge := CLK;

(* revision history
hm	4. aug 2006		rev 1.0
	original version

hm	27. dec 2007	rev 1.1
	changed code for better performance

hm	30. oct. 2008	rev 1.2
	optimized performance
*)
(*@KEY@: END_WORKSHEET *)
END_FUNCTION_BLOCK

(* ---- FF_JKE.ST ---- *)
(*@PROPERTIES_EX@
TYPE: POU
LOCALE: 0
IEC_LANGUAGE: ST
PLC_TYPE: independent
PROC_TYPE: independent
GROUP: LOGIC.FF_EDGE_TRIGGERED
*)
(*@KEY@:DESCRIPTION*)
version 1.2	30. oct. 2008
programmer 	hugo
tested by	oscat

JK-type flip flop with set, reset and rising clock trigger
set and reset are asynchron while the FF is rising edge triggered
J=0 and K=0 and CLK >>> no action
J=1 and K=0 and CLK >>> output = 1
J=0 and K=1 and CLK >>> output = 0
J=1 and K=1 and CLK >>> toggle output
(*@KEY@:END_DESCRIPTION*)
FUNCTION_BLOCK FF_JKE

(*Group:Default*)

VAR_INPUT
	SET :	BOOL;
	J :	BOOL;
	CLK :	BOOL;
	K :	BOOL;
	RST :	BOOL;
END_VAR

VAR_OUTPUT
	Q :	BOOL;
END_VAR

VAR
	edge :	BOOL;
END_VAR

(*@KEY@: WORKSHEET
NAME: FF_JKE
IEC_LANGUAGE: ST
*)
IF rst OR set THEN
	Q := NOT rst;
ELSIF clk AND NOT edge THEN
	IF J XOR K THEN Q := J;
	ELSE Q := K XOR Q;
	END_IF;
END_IF;
edge := CLK;

(* revision history
hm	4. aug 2006		rev 1.0
	original version

hm	27. dec 2007	rev 1.1
	changed code for better performance

hm	30. oct. 2008	rev 1.2
	optimized performance
*)
(*@KEY@: END_WORKSHEET *)
END_FUNCTION_BLOCK

(* ---- FF_RSE.ST ---- *)
(*@PROPERTIES_EX@
TYPE: POU
LOCALE: 0
IEC_LANGUAGE: ST
PLC_TYPE: independent
PROC_TYPE: independent
GROUP: LOGIC.FF_EDGE_TRIGGERED
*)
(*@KEY@:DESCRIPTION*)
version 1.0	16. jul. 2008
programmer 	hugo
tested by	oscat

this is a rising edge triggered rs flip flop
a rising edge on CS sets Q = TRUE and a rising edge on CR sets Q = FALSE.
CR has priority over CS.
(*@KEY@:END_DESCRIPTION*)
FUNCTION_BLOCK FF_RSE

(*Group:Default*)

VAR_INPUT
	CS :	BOOL;
	CR :	BOOL;
	RST :	BOOL;
END_VAR

VAR_OUTPUT
	Q :	BOOL;
END_VAR

VAR
	es :	BOOL;
	er :	BOOL;
END_VAR

(*@KEY@: WORKSHEET
NAME: FF_RSE
IEC_LANGUAGE: ST
*)
IF rst THEN
	(* asynchronous reset *)
	Q := FALSE;
ELSIF CR AND NOT er THEN
	(* rising edge on CR *)
	Q := FALSE;
ELSIF CS AND NOT es THEN
	(* rising edge on CS *)
	Q := TRUE;
END_IF;

es := CS;
er := CR;

(* revision history

hm	16. jul. 2008	rev 1.0
	original version

*)
(*@KEY@: END_WORKSHEET *)
END_FUNCTION_BLOCK

(* ---- FIFO_16.ST ---- *)
(*@PROPERTIES_EX@
TYPE: POU
LOCALE: 0
IEC_LANGUAGE: ST
PLC_TYPE: independent
PROC_TYPE: independent
GROUP: LOGIC.MEMORY
*)
(*@KEY@:DESCRIPTION*)
version 2.0	24. jul. 2009
programmer 	hugo
tested by	oscat

16 Dword FIFO memory
(*@KEY@:END_DESCRIPTION*)
FUNCTION_BLOCK FIFO_16

(*Group:Default*)

VAR_INPUT
	DIN :	DWORD;
	E :	BOOL := TRUE;
	RD :	BOOL;
	WD :	BOOL;
	RST :	BOOL;
END_VAR

VAR_OUTPUT
	DOUT :	DWORD;
	EMPTY :	BOOL := TRUE;
	FULL :	BOOL;
END_VAR

VAR
	fifo :	oscat_ardw_0_15;
	pr :	INT;
	pw :	INT;
END_VAR

(*@KEY@: WORKSHEET
NAME: FIFO_16
IEC_LANGUAGE: ST
*)
IF RST THEN
	pw := pr;
	FULL := FALSE;
	EMPTY := TRUE;
	Dout := DWORD#0;
ELSIF E THEN
	IF NOT EMPTY AND RD THEN
		Dout := fifo[pr];
		pr := INC1(pr,16);
		EMPTY := pr = pw;
		FULL := FALSE;
	END_IF;
	IF NOT FULL AND WD THEN
		fifo[pw] := Din;
		pw := INC1(pw,16);
		FULL := pw = pr;
		EMPTY := FALSE;
	END_IF;
END_IF;

(* revision history

hm	4. aug. 2006	rev 1.0
	original version

hm	19. feb 2008	rev 1.1
	performance improvements

hm	17. oct. 2008	rev 1.2
	improved performance

ks	27. oct. 2008	rev 1.3
	optimized coding

hm	14. mar. 2009	rev 1.4
	removed double assignments

hm 24. jul. 2009	rev 2.0
	chaged inputs E and WR to E, WD and WR
	allow read and write in one cycle

*)

(*@KEY@: END_WORKSHEET *)
END_FUNCTION_BLOCK

(* ---- FIFO_32.ST ---- *)
(*@PROPERTIES_EX@
TYPE: POU
LOCALE: 0
IEC_LANGUAGE: ST
PLC_TYPE: independent
PROC_TYPE: independent
GROUP: LOGIC.MEMORY
*)
(*@KEY@:DESCRIPTION*)
version 2.0	24. jul. 2009
programmer 	hugo
tested by	oscat

32 Dword FIFO memory
(*@KEY@:END_DESCRIPTION*)
FUNCTION_BLOCK FIFO_32

(*Group:Default*)

VAR_INPUT
	DIN :	DWORD;
	E :	BOOL := TRUE;
	RD :	BOOL;
	WD :	BOOL;
	RST :	BOOL;
END_VAR

VAR_OUTPUT
	DOUT :	DWORD;
	EMPTY :	BOOL := TRUE;
	FULL :	BOOL;
END_VAR

VAR
	fifo :	oscat_ardw_0_31;
	pr :	INT;
	pw :	INT;
END_VAR

(*@KEY@: WORKSHEET
NAME: FIFO_32
IEC_LANGUAGE: ST
*)
IF RST THEN
	pw := pr;
	FULL := FALSE;
	EMPTY := TRUE;
	Dout := DWORD#0;
ELSIF E THEN
	IF NOT EMPTY AND RD THEN
		Dout := fifo[pr];
		pr := INC1(pr,32);
		EMPTY := pr = pw;
		FULL := FALSE;
	END_IF;
	IF NOT FULL AND WD THEN
		fifo[pw] := Din;
		pw := INC1(pw,32);
		FULL := pw = pr;
		EMPTY := FALSE;
	END_IF;
END_IF;

(* revision history
hm	4. aug. 2006	rev 1.0
	original version

hm	19. feb 2008	rev 1.1
	performance improvements

hm	17. oct. 2008	rev 1.2
	improved performance

ks	27. oct. 2008 rev 1.3
	improved code

hm	14. mar. 2009	rev 1.4
	removed double assignments

hm 24. jul. 2009	rev 2.0
	chaged inputs E and WR to E, WD and WR
	allow read and write in one cycle

*)

(*@KEY@: END_WORKSHEET *)
END_FUNCTION_BLOCK

(* ---- FILL.ST ---- *)
(*@PROPERTIES_EX@
TYPE: POU
LOCALE: 0
IEC_LANGUAGE: ST
PLC_TYPE: independent
PROC_TYPE: independent
GROUP: STRINGS
*)
(*@KEY@:DESCRIPTION*)
version 1.1	17. dec. 2008
programmer 	hugo
tested by	tobias

the function fill creates a string at length L of characters C.
(*@KEY@:END_DESCRIPTION*)
FUNCTION_BLOCK FILL

(*Group:Default*)

VAR_INPUT
	C :	BYTE;
	L :	INT;
END_VAR

VAR_OUTPUT
	FILL :	STRING;
END_VAR

VAR
	N :	BYTE;
	I :	INT;
	sx :	STRING;
	CHR_TO_STRING :	CHR_TO_STRING;
	FILL_tmp :	STRING;
END_VAR

(*@KEY@: WORKSHEET
NAME: FILL
IEC_LANGUAGE: ST
*)
CHR_TO_STRING(C:=c);
Sx:=CHR_TO_STRING.CHR_TO_STRING;
(* create string *)
N := INT_TO_BYTE(LIMIT(0,L,80));
(* create a string of characters to be connected to str *)
FILL := '';
FOR i := 1 TO 8 DO
    FILL_tmp := FILL;
	FILL := CONCAT(FILL_tmp,FILL);
	IF BIT_OF_DWORD(BYTE_TO_DWORD(N),7) THEN FILL := CONCAT(FILL,Sx); END_IF;
	N := SHL_BYTE(N,1);
END_FOR;

(* revision histroy
hm	29. mar. 2008	rev 1.0
	original release

hm	17. dec. 2008	rev 1.1
	changed function chr to chr_to_string

*)
(*@KEY@: END_WORKSHEET *)
END_FUNCTION_BLOCK

(* ---- FILTER_DW.ST ---- *)
(*@PROPERTIES_EX@
TYPE: POU
LOCALE: 0
IEC_LANGUAGE: ST
PLC_TYPE: independent
PROC_TYPE: independent
GROUP: ENGINEERING.SIGNAL_PROCESSING
*)
(*@KEY@:DESCRIPTION*)
ersion 1.1	3. nov. 2008
programmer 	hugo
tested by	oscat

FILTER_DW is an low pass filter with a programmable time T used for DWORD format.
(*@KEY@:END_DESCRIPTION*)
FUNCTION_BLOCK FILTER_DW

(*Group:Default*)

VAR_INPUT
	X :	DWORD;
	T :	TIME;
END_VAR

VAR_OUTPUT
	Y :	DWORD;
END_VAR

VAR
	last :	UDINT;
	tx :	UDINT;
	init :	BOOL;
	Yi :	REAL;
	T_PLC_MS :	T_PLC_MS;
END_VAR

(*@KEY@: WORKSHEET
NAME: FILTER_DW
IEC_LANGUAGE: ST
*)
(* read system_time *)
T_PLC_MS();
tx:= T_PLC_MS.T_PLC_MS;

(* startup initialisation *)
IF NOT init OR T = t#0s THEN
	init := TRUE;
	Yi := _DWORD_TO_REAL(X);
ELSE
	Yi := Yi + (_DWORD_TO_REAL(X) - _DWORD_TO_REAL(Y)) * UDINT_TO_REAL(tx - last) / TIME_TO_REAL(T);
END_IF;
last := tx;

Y := _REAL_TO_DWORD(Yi);

(*
hm 10. oct. 2008	rev 1.0
	original version

hm	3. nov. 2008	REV 1.1
	corrected an overflow problem
*)
(*@KEY@: END_WORKSHEET *)
END_FUNCTION_BLOCK

(* ---- FILTER_I.ST ---- *)
(*@PROPERTIES_EX@
TYPE: POU
LOCALE: 0
IEC_LANGUAGE: ST
PLC_TYPE: independent
PROC_TYPE: independent
GROUP: ENGINEERING.SIGNAL_PROCESSING
*)
(*@KEY@:DESCRIPTION*)
version 1.0	8. nov. 2008
programmer 	hugo
tested by	oscat

FILTER_I is a low pass filter with a programmable time T used for INT format.
(*@KEY@:END_DESCRIPTION*)
FUNCTION_BLOCK FILTER_I

(*Group:Default*)

VAR_INPUT
	X :	INT;
	T :	TIME;
END_VAR

VAR_OUTPUT
	Y :	INT;
END_VAR

VAR
	Yi :	DINT;
	last :	UDINT;
	tx :	UDINT;
	init :	BOOL;
	T_PLC_MS :	T_PLC_MS;
END_VAR

(*@KEY@: WORKSHEET
NAME: FILTER_I
IEC_LANGUAGE: ST
*)
(* read system time *)
T_PLC_MS();
tx:= T_PLC_MS.T_PLC_MS;

(* startup initialisation *)
IF NOT init OR T = t#0s THEN
	init := TRUE;
	Yi := INT_TO_DINT(X) * DINT#1000;
ELSE
	(* to increase accuracy of the filter we calculate internal Yi wich is Y * 1000 *)
	Yi := Yi + INT_TO_DINT(X - Y) * UDINT_TO_DINT(tx - last) * DINT#1000 / TIME_TO_DINT(T);
END_IF;
last := tx;
Y := DINT_TO_INT(yi / DINT#1000);

(*
hm 8. nov. 2008	rev 1.0
	original version

*)
(*@KEY@: END_WORKSHEET *)
END_FUNCTION_BLOCK

(* ---- FILTER_MAV_DW.ST ---- *)
(*@PROPERTIES_EX@
TYPE: POU
LOCALE: 0
IEC_LANGUAGE: ST
PLC_TYPE: independent
PROC_TYPE: independent
GROUP: ENGINEERING.SIGNAL_PROCESSING
*)
(*@KEY@:DESCRIPTION*)
version 1.3	23. feb. 2009
programmer 	hugo
tested by	oscat

FILTER_MAV_DW is a moving average filter with programmable length N for DWORD Data.
(*@KEY@:END_DESCRIPTION*)
FUNCTION_BLOCK FILTER_MAV_DW

(*Group:Default*)

VAR_INPUT
	X :	DWORD;
	N :	UINT;
	RST :	BOOL;
END_VAR

VAR_OUTPUT
	Y :	DWORD;
END_VAR

VAR
	init :	BOOL;
	buffer :	oscat_ardw_0_31;
	i :	INT;
	tmp :	INT;
END_VAR

(*@KEY@: WORKSHEET
NAME: FILTER_MAV_DW
IEC_LANGUAGE: ST
*)
(* limit N to size of buffer *)
N := MIN(N, UINT#32);

(* startup initialisation *)
IF NOT init OR rst OR N = UINT#0 THEN
	init := TRUE;
	tmp := UINT_TO_INT(N)-1;
	FOR i := 0 TO tmp DO
		buffer[i] := X;
	END_FOR;
	Y := X;
ELSE
	tmp := UINT_TO_INT(N);
	i := INC1(i, tmp);
	Y := UDINT_TO_DWORD(DWORD_TO_UDINT(Y) + (DWORD_TO_UDINT(X) - DWORD_TO_UDINT(buffer[i])) / UINT_TO_UDINT(N));
	buffer[i] := X;
END_IF;

(*
hm 13. oct. 2008	rev 1.0
	original version

hm	27. oct. 2008	rev 1.1
	added typecast to avoid warnings

hm	24. nov. 2008	rev 1.2
	added typecasts to avoid warnings
	avoid divide by 0 if N = 0

hm	23. feb. 2009	rev 1.3
	limit N to max array size

*)
(*@KEY@: END_WORKSHEET *)
END_FUNCTION_BLOCK

(* ---- FILTER_MAV_W.ST ---- *)
(*@PROPERTIES_EX@
TYPE: POU
LOCALE: 0
IEC_LANGUAGE: ST
PLC_TYPE: independent
PROC_TYPE: independent
GROUP: ENGINEERING.SIGNAL_PROCESSING
*)
(*@KEY@:DESCRIPTION*)
version 1.4	26. MAR. 2011
programmer 	    hugo
tested by		oscat

FILTER_MAV_W is a moving average filter with programmable length N for WORD Data.

(*@KEY@:END_DESCRIPTION*)
FUNCTION_BLOCK FILTER_MAV_W

(*Group:Default*)

VAR_INPUT
	X :	WORD;
	N :	UINT;
	RST :	BOOL;
END_VAR

VAR_OUTPUT
	Y :	WORD;
END_VAR

VAR
	init :	BOOL;
	buffer :	oscat_FILTER_MAV_W;
	i :	INT;
	sum :	UDINT;
	tmp :	INT;
END_VAR

(*@KEY@: WORKSHEET
NAME: FILTER_MAV_W
IEC_LANGUAGE: ST
*)
(* limit N to size of buffer *)
N := MIN(N, UINT#32);

(* startup initialisation *)
IF NOT init OR rst OR N = UINT#0 THEN
	init := TRUE;
	tmp := UINT_TO_INT(N) - 1;
	FOR i := 1 TO tmp DO
		buffer[i] := X;
	END_FOR;
	sum := UINT_TO_UDINT(WORD_TO_UINT(Y) * N);
	Y := X;
ELSE
	tmp := UINT_TO_INT(N);
	i := INC1(i, tmp);
	sum := sum + WORD_TO_UDINT(X) - WORD_TO_UDINT(buffer[i]);
	Y := UDINT_TO_WORD(sum / UINT_TO_UDINT(N));
	buffer[i] := X;
END_IF;

(*
hm 13. oct. 2008	rev 1.0
	original version

hm	18. oct. 2008	rev 1.1
	added typecast to avoid warnings

hm	24. nov. 2008	rev 1.2
	added typecasts to avoid warnings
	avoid devide by 0 if N = 0

hm	23. feb. 2009	rev 1.3
	limit N to max array size

hm	26. mar. 2011	rev 1.4
	corrected error in calculation
*)

(*@KEY@: END_WORKSHEET *)
END_FUNCTION_BLOCK

(* ---- FILTER_W.ST ---- *)
(*@PROPERTIES_EX@
TYPE: POU
LOCALE: 0
IEC_LANGUAGE: ST
PLC_TYPE: independent
PROC_TYPE: independent
GROUP: ENGINEERING.SIGNAL_PROCESSING
*)
(*@KEY@:DESCRIPTION*)
version 1.2	25. jan. 2011
programmer 	hugo
tested by	oscat

FILTER_W is an low pass filter with a programmable time T used for WORD format.
(*@KEY@:END_DESCRIPTION*)
FUNCTION_BLOCK FILTER_W

(*Group:Default*)

VAR_INPUT
	X :	WORD;
	T :	TIME;
END_VAR

VAR_OUTPUT
	Y :	WORD;
END_VAR

VAR
	last :	UDINT;
	tx :	UDINT;
	init :	BOOL;
	tmp :	DINT;
	T_PLC_MS :	T_PLC_MS;
END_VAR

(*@KEY@: WORKSHEET
NAME: FILTER_W
IEC_LANGUAGE: ST
*)
(* read system time *)
T_PLC_MS();
tx:= T_PLC_MS.T_PLC_MS;

(* startup initialisation *)
IF NOT init OR T = T#0s THEN
	init := TRUE;
	last := tx;
	Y := X;
ELSIF Y = X THEN
	last := tx;
ELSE
	tmp := UINT_TO_DINT(WORD_TO_UINT(X) - WORD_TO_UINT(Y)) * UDINT_TO_DINT(tx - last) / TIME_TO_DINT(T);
	IF tmp <> DINT#0 THEN
		Y := DINT_TO_WORD(WORD_TO_DINT(Y) + tmp);
		last := tx;
	END_IF;
END_IF;

(*
hm 10. oct. 2008	rev 1.0
	original version

hm	3. nov. 2008	rev 1.1
	fixed overflow problem in formula

hm	25. jan. 2011	rev 1.2
	fixed error in formula
*)
(*@KEY@: END_WORKSHEET *)
END_FUNCTION_BLOCK

(* ---- FILTER_WAV.ST ---- *)
(*@PROPERTIES_EX@
TYPE: POU
LOCALE: 0
IEC_LANGUAGE: ST
PLC_TYPE: independent
PROC_TYPE: independent
GROUP: ENGINEERING.SIGNAL_PROCESSING
*)
(*@KEY@:DESCRIPTION*)
version 1.2	10. mar. 2009
programmer 	hugo
tested by	oscat

FILTER_WAV is a moving average filter with programmable length N for DWORD Data.

(*@KEY@:END_DESCRIPTION*)
FUNCTION_BLOCK FILTER_WAV

(*Group:Default*)

VAR_INPUT
	X :	REAL;
	W :	oscat_arr_0_15;
	RST :	BOOL;
END_VAR

VAR_OUTPUT
	Y :	REAL;
END_VAR

VAR
	init :	BOOL;
	buffer :	oscat_arr_0_15;
	i :	INT;
	n :	INT;
END_VAR

(*@KEY@: WORKSHEET
NAME: FILTER_WAV
IEC_LANGUAGE: ST
*)
(* startup initialisation *)
IF NOT init OR rst THEN
	init := TRUE;
	FOR i := 0 TO 15 DO
		buffer[i] := X;
	END_FOR;
	i := 15;
	Y := X;
ELSE
	i := INC1(i, 16);
	buffer[i] := X;
END_IF;

(* calculate the weighted average *)
Y := 0.0;
FOR n := 0 TO 15 DO
	Y := buffer[i] * W[n] + Y;
	i := DEC1(i, 16);
END_FOR;

(*
hm 	14. oct. 2008	rev 1.0
	original version

hm	27. oct. 2008	rev 1.1
	changed _DEC and _INC to DEC1 and INC1

hm	10. mar. 2009	rev 1.2
	real constants updated to new systax using dot

*)

(*@KEY@: END_WORKSHEET *)
END_FUNCTION_BLOCK

(* ---- FIND_CHAR.ST ---- *)
(*@PROPERTIES_EX@
TYPE: POU
LOCALE: 0
IEC_LANGUAGE: ST
PLC_TYPE: independent
PROC_TYPE: independent
GROUP: STRINGS
*)
(*@KEY@:DESCRIPTION*)
version 1.3	21. oct. 2008
programmer 	hugo
tested by	tobias

find_char searches str and returns the starting position of the first character that is not a control character.
control characters are the ascii character 00 .. 31 and 127
(*@KEY@:END_DESCRIPTION*)
FUNCTION_BLOCK FIND_CHAR

(*Group:Default*)

VAR_INPUT
	STR :	STRING;
	POS :	INT;
END_VAR

VAR_OUTPUT
	FIND_CHAR :	INT;
END_VAR

VAR
	EXT_ASCII :	BOOL;
	X :	INT;
	stop :	INT;
	i :	INT;
END_VAR

(*@KEY@: WORKSHEET
NAME: FIND_CHAR
IEC_LANGUAGE: ST
*)
EXT_ASCII := SETUP_EXTENDED_ASCII(FALSE);

stop := LEN(str);
FOR i := MAX(pos,1) TO stop DO;
    X := GET_CHAR(str,i);
	IF X > 31 AND ((EXT_ASCII AND X <> 127) OR (NOT EXT_ASCII AND X < 127)) THEN
		FIND_CHAR := i;
		RETURN;
	END_IF;
END_FOR;
FIND_CHAR := 0;

(* revision history
hm	29. feb 2008	rev 1.0
	original version

hm	26. mar. 2008	rev 1.1
	char will now accept extended ascii

hm	29. mar. 2008	rev 1.2
	changed STRING to STRING(STRING_LENGTH)

hm	19. oct. 2008	rev 1.3
	changes setup constants
*)
(*@KEY@: END_WORKSHEET *)
END_FUNCTION_BLOCK

(* ---- FIND_CTRL.ST ---- *)
(*@PROPERTIES_EX@
TYPE: POU
LOCALE: 0
IEC_LANGUAGE: ST
PLC_TYPE: independent
PROC_TYPE: independent
GROUP: STRINGS
*)
(*@KEY@:DESCRIPTION*)
version 1.2	29. mar. 2008
programmer 	hugo
tested by	tobias

find_ctrl searches str and returns the starting position of a control character
control characters are the ascii character 00 .. 31 and 127.
(*@KEY@:END_DESCRIPTION*)
FUNCTION_BLOCK FIND_CTRL

(*Group:Default*)

VAR_INPUT
	STR :	STRING;
	POS :	INT;
END_VAR

VAR_OUTPUT
	FIND_CTRL :	INT;
END_VAR

VAR
	x :	INT;
	stop :	INT;
	i :	INT;
END_VAR

(*@KEY@: WORKSHEET
NAME: FIND_CTRL
IEC_LANGUAGE: ST
*)
stop := LEN(str);
FOR i := MAX(pos,1) TO stop DO;
    x := GET_CHAR(str,i);
	IF (x < 32) OR (x = 127) THEN
		FIND_CTRL := i;
		RETURN;
	END_IF;
END_FOR;
FIND_CTRL := 0;

(* revision history
hm	29. feb 2008	rev 1.0
	original version

hm	26. mar. 2008	rev 1.1
	character 127 is now recognized as control

hm	29. mar. 2008	rev 1.2
	changed STRING to STRING(STRING_LENGTH)
*)
(*@KEY@: END_WORKSHEET *)
END_FUNCTION_BLOCK

(* ---- FIND_NONUM.ST ---- *)
(*@PROPERTIES_EX@
TYPE: POU
LOCALE: 0
IEC_LANGUAGE: ST
PLC_TYPE: independent
PROC_TYPE: independent
GROUP: STRINGS
*)
(*@KEY@:DESCRIPTION*)
version 1.3	21. oct. 2008
programmer 	hugo
tested by	tobias

find_noNum searches str and returns the first position which is not a number.
a number is characterized by a letter "0..9" or "."
(*@KEY@:END_DESCRIPTION*)
FUNCTION_BLOCK FIND_NONUM

(*Group:Default*)

VAR_INPUT
	STR :	STRING;
	POS :	INT;
END_VAR

VAR_OUTPUT
	FIND_NONUM :	INT;
END_VAR

VAR
	X :	INT;
	end :	INT;
END_VAR

(*@KEY@: WORKSHEET
NAME: FIND_NONUM
IEC_LANGUAGE: ST
*)
end := LEN(str);
FOR pos := MAX(pos,1) TO LEN(str) DO;
     X :=GET_CHAR(str,pos);
	IF (X < 48 AND X <> 46) OR X > 57 THEN
		find_nonum := pos;
		RETURN;
	END_IF;
END_FOR;
find_nonum := 0;

(* revision history
hm	6. oct. 2006	rev 1.0
	original version

hm	29. feb 2008	rev 1.1
	added input pos to start search at position

hm	29. mar. 2008	rev 1.2
	changed STRING to STRING(STRING_LENGTH)

hm	21. oct. 2008	rev 1.3
	optimized code

*)
(*@KEY@: END_WORKSHEET *)
END_FUNCTION_BLOCK

(* ---- FIND_NUM.ST ---- *)
(*@PROPERTIES_EX@
TYPE: POU
LOCALE: 0
IEC_LANGUAGE: ST
PLC_TYPE: independent
PROC_TYPE: independent
GROUP: STRINGS
*)
(*@KEY@:DESCRIPTION*)
version 1.2	29. mar. 2008
programmer 	hugo
tested by	tobias

find_Num searches str and returns the starting position of a number
a number is characterized by a letter "0..9" or "."
(*@KEY@:END_DESCRIPTION*)
FUNCTION_BLOCK FIND_NUM

(*Group:Default*)

VAR_INPUT
	STR :	STRING;
	POS :	INT;
END_VAR

VAR_OUTPUT
	FIND_NUM :	INT;
END_VAR

VAR
	X :	INT;
	stop :	INT;
END_VAR

(*@KEY@: WORKSHEET
NAME: FIND_NUM
IEC_LANGUAGE: ST
*)
stop := LEN(str);
FOR pos := MAX(pos,1) TO stop DO;
    X :=GET_CHAR(str,pos);
	IF (X > 47 AND X < 58) OR X = 46 THEN
		find_num := pos;
		RETURN;
	END_IF;
END_FOR;
find_num := 0;

(* revision history
hm	6. oct. 2006	rev 1.0
	original version

hm	29. feb 2008	rev 1.1
	added input pos to start search at position

hm	29. mar. 2008	rev 1.2
	changed STRING to STRING(STRING_LENGTH)

*)
(*@KEY@: END_WORKSHEET *)
END_FUNCTION_BLOCK

(* ---- FINDB.ST ---- *)
(*@PROPERTIES_EX@
TYPE: POU
LOCALE: 0
IEC_LANGUAGE: ST
PLC_TYPE: independent
PROC_TYPE: independent
GROUP: STRINGS
*)
(*@KEY@:DESCRIPTION*)
version 1.3	29. mar. 2008
programmer 	hugo
tested by	tobias

the function find searches an str1 for the presence of str2 and returns the first position of str1 of the last presence in instring.
the function is similar to find except it searches from the right to left.
 a 0 is returned if the string is not found.
(*@KEY@:END_DESCRIPTION*)
FUNCTION_BLOCK FINDB

(*Group:Default*)

VAR_INPUT
	STR1 :	oscat_STRING250;
	STR2 :	STRING;
END_VAR

VAR_OUTPUT
	FINDB :	INT;
END_VAR

VAR
	pos :	INT;
	length :	INT;
	string_temp :	oscat_STRING250;
END_VAR

(*@KEY@: WORKSHEET
NAME: FINDB
IEC_LANGUAGE: ST
*)
length := LEN(str2);
pos := LEN(str1) - length +1;
WHILE (pos >= 1) DO
    string_temp := MID(str1,length,pos);
    IF EQ_STRING(string_temp,str2) THEN
		FindB := pos;
		RETURN;
	END_IF;
pos := pos -1;
END_WHILE;
FindB := 0;

(* revision history
hm	6. oct 2006		rev 1.0
	original version

hm	15 dec 2007		rev 1.1
	changed code for better performance

hm	29. feb 2008	rev 1.2
	added findb := 0 for compatibility reasons

hm	29. mar. 2008	rev 1.3
	changed STRING to STRING(STRING_LENGTH)
*)
(*@KEY@: END_WORKSHEET *)
END_FUNCTION_BLOCK

(* ---- FINDB_NONUM.ST ---- *)
(*@PROPERTIES_EX@
TYPE: POU
LOCALE: 0
IEC_LANGUAGE: ST
PLC_TYPE: independent
PROC_TYPE: independent
GROUP: STRINGS
*)
(*@KEY@:DESCRIPTION*)
version 1.3	21. oct. 2008
programmer 	hugo
tested by	oscat

findB_noNum searches str backwards and returns the last position which is not a number.
a number is characterized by a letter "0..9" or "."
(*@KEY@:END_DESCRIPTION*)
FUNCTION_BLOCK FINDB_NONUM

(*Group:Default*)

VAR_INPUT
	STR :	STRING;
END_VAR

VAR_OUTPUT
	FINDB_NONUM :	INT;
END_VAR

VAR
	pos :	INT;
	x :	INT;
END_VAR

(*@KEY@: WORKSHEET
NAME: FINDB_NONUM
IEC_LANGUAGE: ST
*)
pos := LEN(str);
WHILE (pos >=1) DO
    x :=GET_CHAR(str,pos);
	IF (X < 48 AND X <> 46) OR X > 57 THEN
		findB_nonum := pos;
		RETURN;
	END_IF;
pos := pos -1;
END_WHILE;
findB_nonum := 0;

(* revision history
hm	6. oct 2006		rev 1.0
	original version

hm	29. feb 2008	rev 1.1
	improved performance

hm	29. mar. 2008	rev 1.2
	changed STRING to STRING(STRING_LENGTH)

hm	21. oct. 2008	rev 1.3
	optimized code
*)
(*@KEY@: END_WORKSHEET *)
END_FUNCTION_BLOCK

(* ---- FINDB_NUM.ST ---- *)
(*@PROPERTIES_EX@
TYPE: POU
LOCALE: 0
IEC_LANGUAGE: ST
PLC_TYPE: independent
PROC_TYPE: independent
GROUP: STRINGS
*)
(*@KEY@:DESCRIPTION*)
version 1.2	29. mar. 2008
programmer 	hugo
tested by	tobias

findB_Num searches str backward and returns the last position of a number
a number is characterized by a letter "0..9" or "."
(*@KEY@:END_DESCRIPTION*)
FUNCTION_BLOCK FINDB_NUM

(*Group:Default*)

VAR_INPUT
	STR :	STRING;
END_VAR

VAR_OUTPUT
	FINDB_NUM :	INT;
END_VAR

VAR
	pos :	INT;
	x :	INT;
END_VAR

(*@KEY@: WORKSHEET
NAME: FINDB_NUM
IEC_LANGUAGE: ST
*)
findB_num := 0;
pos := LEN(str);
WHILE (pos >=1) DO
    x :=GET_CHAR(str,pos);
	IF (x > 47 AND x < 58) OR x = 46 THEN
		findB_num := pos;
		RETURN;
	END_IF;
pos := pos -1;
END_WHILE;

(* revision history
hm	6. oct 2006		rev 1.0
	original version

hm	29. feb 2008	rev 1.1
	improved performance

hm	29. mar. 2008	rev 1.2
	changed STRING to STRING(STRING_LENGTH)
*)
(*@KEY@: END_WORKSHEET *)
END_FUNCTION_BLOCK

(* ---- FINDP.ST ---- *)
(*@PROPERTIES_EX@
TYPE: POU
LOCALE: 0
IEC_LANGUAGE: ST
PLC_TYPE: independent
PROC_TYPE: independent
GROUP: STRINGS
*)
(*@KEY@:DESCRIPTION*)
version 1.2	29. mar. 2008
programmer 	hugo
tested by	tobias

the function findP searches a string str for the occurence of src beginning at the position pos.
(*@KEY@:END_DESCRIPTION*)
FUNCTION_BLOCK FINDP

(*Group:Default*)

VAR_INPUT
	STR :	STRING;
	SRC :	STRING;
	POS :	INT;
END_VAR

VAR_OUTPUT
	FINDP :	INT;
END_VAR

VAR
	i :	INT;
	ls :	INT;
	lx :	INT;
	stp :	INT;
	st_tmp :	STRING;
END_VAR

(*@KEY@: WORKSHEET
NAME: FINDP
IEC_LANGUAGE: ST
*)
ls := LEN(str);
lx := LEN(src);
IF ls < lx OR lx = 0 THEN RETURN; END_IF;
stp := ls - lx + 1;
FOR i := MAX(pos,1) TO stp DO
    st_tmp := MID(str,lx,i);
	IF EQ_STRING(st_tmp,src) THEN
		FINDP := i;
		RETURN;
	END_IF;
END_FOR;
FINDP := 0;

(* revision histroy
hm	4. feb. 2008	rev 1.0
	original release

hm	29. feb 2008	rev 1.1
	ADDED MAX(pos,1) in loop initialization

hm	29. mar. 2008	rev 1.2
	changed STRING to STRING(STRING_LENGTH)
*)
(*@KEY@: END_WORKSHEET *)
END_FUNCTION_BLOCK

(* ---- FIX.ST ---- *)
(*@PROPERTIES_EX@
TYPE: POU
LOCALE: 0
IEC_LANGUAGE: ST
PLC_TYPE: independent
PROC_TYPE: independent
GROUP: STRINGS
*)
(*@KEY@:DESCRIPTION*)
version 1.0	29. mar. 2008
programmer 	hugo
tested by	tobias

the function fix truncates a string at length L
or if the string is shorter then L it will be filled with ending Spaces till its length = N.
(*@KEY@:END_DESCRIPTION*)
FUNCTION_BLOCK FIX

(*Group:Default*)

VAR_INPUT
	STR :	oscat_STRING250;
	L :	INT;
	C :	BYTE;
	M :	INT;
END_VAR

VAR_OUTPUT
	FIX :	oscat_STRING250;
END_VAR

VAR
	N :	INT;
	FILL :	FILL;
END_VAR

(*@KEY@: WORKSHEET
NAME: FIX
IEC_LANGUAGE: ST
*)
(* make sure L does not exceed the limits of a string *)
N := LIMIT(0,L,255) - LEN(str);
IF N <= 0 THEN
	(* truncate the string at length N *)
	IF M = 1 THEN
		FIX := RIGHT(str,L);
	ELSE
		FIX := LEFT(str,L);
	END_IF;
ELSIF M = 1 THEN
	(* connect fill characters at the beginning *)
    FILL(C:=C,L:=N);
	FIX := CONCAT(FILL.FILL,str);
ELSIF M = 2 THEN
	(* center str beween fill characters *)
	(* for an uneven number of fill characters, there is one more at the end *)
    FILL(C:=C,L:=_BYTE_TO_INT(SHR_BYTE(INT_TO_BYTE(N+1),1)));
	FIX := CONCAT(str,FILL.FILL);
    FILL(C:=C,L:=_BYTE_TO_INT(SHR_BYTE(INT_TO_BYTE(N),1)));
	FIX := CONCAT(FILL.FILL,FIX);
ELSE
	(* connect fill characters at the end *)
    FILL(C:=C,L:=N);
	FIX := CONCAT(str,FILL.FILL);
END_IF;

(* revision histroy
hm	29. mar. 2008	rev 1.0
	original release

*)
(*@KEY@: END_WORKSHEET *)
END_FUNCTION_BLOCK

(* ---- FLOAT_TO_REAL.ST ---- *)
(*@PROPERTIES_EX@
TYPE: POU
LOCALE: 0
IEC_LANGUAGE: ST
PLC_TYPE: independent
PROC_TYPE: independent
GROUP: STRINGS
*)
(*@KEY@:DESCRIPTION*)
version 1.3	23. oct. 2008
programmer 	hugo
tested by	oscat

FLOAT_TO_REAL converts a string to a REAL.
the function ignores all wrong characters.
the comma can be , or .
the exponent has to start with capital E or lowercase e .
(*@KEY@:END_DESCRIPTION*)
FUNCTION_BLOCK FLOAT_TO_REAL

(*Group:Default*)

VAR_INPUT
	FLT :	oscat_STRING20;
END_VAR

VAR_OUTPUT
	FLOAT_TO_REAL :	REAL;
END_VAR

VAR
	i :	INT;
	X :	BYTE;
	sign :	INT := 1;
	stop :	INT;
	tmp :	DINT;
	d :	INT;
	DEC_TO_INT :	DEC_TO_INT;
	CODE :	CODE;
END_VAR

(*@KEY@: WORKSHEET
NAME: FLOAT_TO_REAL
IEC_LANGUAGE: ST
*)
sign := 1;
d := 0;
stop := LEN(FLT);
tmp := DINT#0;

(* we first check for sign and exit if first number or dot is reached *)
FOR i := 1 TO stop DO
    CODE(STR:=FLT,POS:=i);
    X := CODE.CODE;
	IF X > BYTE#47 AND X < BYTE#58 OR X = BYTE#46 THEN
		EXIT;
	ELSIF X = BYTE#45 THEN
		(* code 45 is sign *)
		sign := -1;
	END_IF;
END_FOR;

(* now we scan numbers till end or dot or E is reached *)
FOR i := i TO stop DO
    CODE(STR:=FLT,POS:=i);
    X := CODE.CODE;
	IF X = BYTE#44 OR X = BYTE#46 OR X = BYTE#69 OR X = BYTE#101 THEN
		EXIT;
	(* calculate the value of the digit *)
	ELSIF X > BYTE#47 AND x < BYTE#58 THEN
		tmp := tmp * DINT#10 + _BYTE_TO_DINT(X) - DINT#48;
	END_IF;
END_FOR;

(* process the portion after the comma if comma or dot is reached exit if exponent starts *)
IF x = BYTE#44 OR X = BYTE#46 THEN
	FOR i := i + 1 TO stop DO
        CODE(STR:=FLT,POS:=i);
        X := CODE.CODE;
		IF X = BYTE#69 OR X = BYTE#101 THEN
			EXIT;
		ELSIF x > BYTE#47 AND x < BYTE#58 THEN
			tmp := tmp * DINT#10 + _BYTE_TO_DINT(X) - DINT#48;
			d := d - 1;
		END_IF;
	END_FOR;
END_IF;

(* process exponent if present *)
IF (X = BYTE#69 OR X = BYTE#101) AND i<=stop THEN
    DEC_TO_INT(DEC:=MID(FLT, MIN(stop - i,10),MIN(stop,i+1)));
    d := d + DEC_TO_INT.DEC_TO_INT;

(*    DEC_TO_INT(DEC:=RIGHT(FLT, MIN(stop - i,10)));
    d := d + DEC_TO_INT.DEC_TO_INT;*)
END_IF;

FLOAT_TO_REAL :=  EXPN(10.0, d) * DINT_TO_REAL(TMP * INT_TO_DINT(SIGN));

(* revision histroy
hm	22. jun. 2008	rev 1.0
	original release

hm	2. oct. 2008	rev 1.1
	fixed an error, characters 8 and 9 would not be converted

hm	22. oct. 2008	rev 1.2
	last fix was not done correctly

hm	23. oct. 2008	rev 1.3
	optimzed code
*)
(*@KEY@: END_WORKSHEET *)
END_FUNCTION_BLOCK

(* ---- FLOW_CONTROL.ST ---- *)
(*@PROPERTIES_EX@
TYPE: POU
LOCALE: 0
IEC_LANGUAGE: ST
PLC_TYPE: independent
PROC_TYPE: independent
GROUP: ENGINEERING.AUTOMATION
*)
(*@KEY@:DESCRIPTION*)
version 1.0	28. jun. 2008
programmer 	hugo
tested by	oscat

FLOW_CONTROL switches a valves depending on the input in.
flow control also limits the maximum ontime of the valve and controls pressure on the output side.
(*@KEY@:END_DESCRIPTION*)
FUNCTION_BLOCK FLOW_CONTROL

(*Group:Default*)

VAR_INPUT
	IN :	BOOL;
	REQ :	BOOL;
	ENQ :	BOOL;
	RST :	BOOL := FALSE;
	T_AUTO :	TIME := T#1h;
	T_DELAY :	TIME := T#23h;
END_VAR

VAR_OUTPUT
	Q :	BOOL;
	STATUS :	BYTE;
END_VAR

VAR
	timer :	TP_1D;
END_VAR

(*@KEY@: WORKSHEET
NAME: FLOW_CONTROL
IEC_LANGUAGE: ST
*)
STATUS := BYTE#100;
IF RST THEN
	Q := FALSE;
	timer(rst := TRUE);
	timer.RST := FALSE;
	STATUS := BYTE#103;
ELSIF ENQ THEN
	IF IN THEN
		status := BYTE#101;
	END_IF;
	IF REQ THEN
		(* timer will generate a timed pulse after TP goes high *)
		timer.PT1 := T_AUTO;
		timer.PTD := T_DELAY;
		timer.IN := TRUE;
		STATUS := BYTE#102;
	END_IF;
END_IF;

(* set output and run timer *)
timer();
timer.IN := FALSE;
Q := (IN AND ENQ) OR timer.Q;

(* revision history
hm 	28. jun. 2008 	rev 1.0
	original version

*)
(*@KEY@: END_WORKSHEET *)
END_FUNCTION_BLOCK

(* ---- FLOW_CONTROL_4.ST ---- *)
(*@PROPERTIES_EX@
TYPE: POU
LOCALE: 0
IEC_LANGUAGE: ST
PLC_TYPE: independent
PROC_TYPE: independent
GROUP: ENGINEERING.AUTOMATION
*)
(*@KEY@:DESCRIPTION*)
version 1.0	19. jun 2008
programmer 	hugo
tested by	oscat

FLOW_CONTROL switches up to 4 valves depending on the 4 inputs i and generates a safety valve signal.
flow control also limits the maximum ontime of valves and controls pressure on the output side.
a diangnostic mode can automatically check all valves for operation and report errors.
anti freeze can be used to protect valves from icing during cold season´.
(*@KEY@:END_DESCRIPTION*)
FUNCTION_BLOCK FLOW_CONTROL_4

(*Group:Default*)

VAR_INPUT
	I0 :	BOOL;
	I1 :	BOOL;
	I2 :	BOOL;
	I3 :	BOOL;
	PR :	BOOL;
	ICE :	BOOL;
	DIAG :	BOOL;
	ENQ :	BOOL;
	RST :	BOOL := FALSE;
	TD_WAIT :	TIME := T#5s;
	TD_S :	TIME := T#10s;
	TD_0 :	TIME := T#10s;
END_VAR

VAR_OUTPUT
	QS :	BOOL;
	Q0 :	BOOL;
	Q1 :	BOOL;
	Q2 :	BOOL;
	Q3 :	BOOL;
	ERROR :	BOOL;
	STATUS :	BYTE;
END_VAR

VAR
	state :	INT;
	timer :	TP;
END_VAR

(*@KEY@: WORKSHEET
NAME: FLOW_CONTROL_4
IEC_LANGUAGE: ST
*)
IF RST THEN
	STATUS := BYTE#100;
	state := 0;
	error := FALSE;

ELSIF DIAG THEN
	(* diag puts pressure by opening QS for TD_wait,
	thencloses all valves and waits for td_wait, opens valve_0 and checks pressure after td_0
	if pressure is too low, an error is present.
	continue the same procedure for all valves *)
	CASE state OF
		0 : (* start diag operation *)
			(* close all valves and pressurize the system *)
			QS := TRUE;
			Q0 := FALSE;
			Q1 := FALSE;
			Q2 := FALSE;
			Q3 := FALSE;
			timer(in := TRUE, pt := TD_WAIT);
			timer.IN := FALSE;
			state := 1;
		1 : (* wait for TD_wait *)
			timer();
			IF NOT timer.Q THEN
				QS := FALSE;
				timer(in := TRUE, pt := TD_S);
				timer.IN := FALSE;
				state := 2;
			END_IF;
		2:	(* wait for safety valve pressure test *)
			timer();
			IF NOT timer.Q THEN
				IF NOT pr THEN
					(* system pressure failure *)
					ERROR := TRUE;
					STATUS := BYTE#1;
					RETURN;
				END_IF;
				timer(in := TRUE, pt := TD_0);
				timer.IN := FALSE;
				Q0 := TRUE;
				state := 3;
			END_IF;
		3:	(* wait for pressure on Q0 to hold TD_0 *)
			timer();
			IF NOT timer.Q THEN
				IF NOT pr THEN
					(* valve 0 pressure failure *)
					ERROR := TRUE;
					STATUS := BYTE#1;
					RETURN;
				END_IF;
				Q0 := FALSE;
				QS := TRUE;
			END_IF;
	END_CASE;
ELSIF ICE THEN
	(* when frost is present we close the safety valve and open all other valves to depressurize the valves *)
	QS := FALSE;
	Q0 := TRUE;
	Q1 := TRUE;
	Q2 := TRUE;
	Q3 := TRUE;
	STATUS := BYTE#110;

ELSIF NOT error AND ENQ THEN
		Q0 := I0;
		Q1 := I1;
		Q2 := I2;
		Q3 := I3;
		QS := Q0 OR Q1 OR Q2 OR Q3;
		STATUS := BYTE#100;

		(* maximum ontime check *)
ELSE
	Q0 := FALSE;
	Q1 := FALSE;
	Q2 := FALSE;
	Q3 := FALSE;
END_IF;

(* revision history
hm 	19. jun. 2008 	rev 1.0
	original version

*)
(*@KEY@: END_WORKSHEET *)
END_FUNCTION_BLOCK

(* ---- FLOW_METER.ST ---- *)
(*@PROPERTIES_EX@
TYPE: POU
LOCALE: 0
IEC_LANGUAGE: ST
PLC_TYPE: independent
PROC_TYPE: independent
GROUP: ENGINEERING.MEASUREMENTS
*)
(*@KEY@:DESCRIPTION*)
version 1.0	23. jan. 2011
programmer 	hugo
tested by	oscat

Flow meter measures flow according to gated time or pulses.
(*@KEY@:END_DESCRIPTION*)
FUNCTION_BLOCK FLOW_METER

(*Group:Default*)

VAR_INPUT
	VX :	REAL;
	E :	BOOL;
	RST :	BOOL;
	PULSE_MODE :	BOOL;
	UPDATE_TIME :	TIME := T#1s;
END_VAR

VAR_OUTPUT
	F :	REAL;
END_VAR

VAR_IN_OUT
	X :	REAL;
	Y :	UDINT;
END_VAR

VAR
	T_PLC_MS :	T_PLC_MS;
	tx :	TIME;
	tl :	TIME;
	int1 :	INTEGRATE;
	init :	BOOL;
	e_last :	BOOL;
	tmp :	INT;
	x_last :	REAL;
	y_last :	UDINT;
END_VAR

(*@KEY@: WORKSHEET
NAME: FLOW_METER
IEC_LANGUAGE: ST
*)
IF NOT init THEN	(* init on power up *)
	init := TRUE;
	tl := tx;
	x_last := X;
	y_last := Y;
	int1.K := 2.7777777777777777E-4;
END_IF;

(* run integrator *)
int1(E := NOT (RST OR PULSE_MODE) AND E, X := VX, Y := X);	(* gated operation *)
X := int1.Y;

IF RST THEN		(* reset *)
	X := 0.0;
	Y := UDINT#0;
	tl := tx;
	x_last := 0.0;
	y_last := UDINT#0;
ELSIF E AND PULSE_MODE THEN	(* check for pulse mode *)
	IF NOT e_last THEN X := X + VX; END_IF;
END_IF;
e_last := E;

(* reduce X to be less than 1 and increase Y respectively *)
IF X > 1.0 THEN
	tmp := FLOOR(X);
	Y := Y + _INT_TO_UDINT(tmp);
	X := X - INT_TO_REAL(tmp);
END_IF;

(* calculate the current flow *)
T_PLC_MS();
tx := UDINT_TO_TIME(T_PLC_MS.T_PLC_MS);
IF tx - tl >= UPDATE_TIME AND UPDATE_TIME > t#0s THEN
	F := (UDINT_TO_REAL(Y - y_last) + X - x_last) / TIME_TO_REAL(tx - tl) * 3.6E6;
	y_last := Y;
	x_last := X;
	tl := tx;
END_IF;

(* revision history
hm	23. jan. 2011	rev 1.0
	original version

*)
(*@KEY@: END_WORKSHEET *)
END_FUNCTION_BLOCK

(* ---- FSTRING_TO_BYTE.ST ---- *)
(*@PROPERTIES_EX@
TYPE: POU
LOCALE: 0
IEC_LANGUAGE: ST
PLC_TYPE: independent
PROC_TYPE: independent
GROUP: STRINGS
*)
(*@KEY@:DESCRIPTION*)
version 1.1	20. sep. 2008
programmer 	hugo
tested by		oscat

FSTRING_TO_BYTE converts a formatted string into a byte.
the string can be of the form 2#01010, 8#7234, 16#2AD3 and 1234
(*@KEY@:END_DESCRIPTION*)
FUNCTION_BLOCK FSTRING_TO_BYTE

(*Group:Default*)

VAR_INPUT
	IN :	oscat_STRING12;
END_VAR

VAR_OUTPUT
	FSTRING_TO_BYTE :	BYTE;
END_VAR

VAR
	CLEAN :	CLEAN;
	BIN_TO_BYTE :	BIN_TO_BYTE;
	OCT_TO_BYTE :	OCT_TO_BYTE;
	HEX_TO_BYTE :	HEX_TO_BYTE;
	tmp :	oscat_STRING3;
END_VAR

(*@KEY@: WORKSHEET
NAME: FSTRING_TO_BYTE
IEC_LANGUAGE: ST
*)
IF LEN(IN)=0 THEN FSTRING_TO_BYTE := BYTE#0;RETURN;END_IF;

tmp := LEFT(IN,MIN(2,LEN(IN)));
IF EQ_STRING(tmp,'2#') THEN
	(* we need to convert binary *)
    BIN_TO_BYTE(BIN:=RIGHT(in, LEN(in) - 2));
	FSTRING_TO_BYTE := BIN_TO_BYTE.BIN_TO_BYTE;
ELSIF EQ_STRING(tmp,'8#') THEN
	(* weneed to convert octals *)
    OCT_TO_BYTE(OCT:=RIGHT(in, LEN(in) - 2));
	FSTRING_TO_BYTE := OCT_TO_BYTE.OCT_TO_BYTE;
ELSE
    tmp := LEFT(IN,MIN(3,LEN(IN)));
    IF EQ_STRING(tmp,'16#') THEN
	    (* we need to convert hexadecimal *)
        HEX_TO_BYTE(HEX:=RIGHT(in, LEN(in) - 3));
	    FSTRING_TO_BYTE := HEX_TO_BYTE.HEX_TO_BYTE;
    ELSE
	    (* we assume decimal representation *)
        CLEAN(IN:=in,CX:='0123456789');
	    FSTRING_TO_BYTE := STRING_TO_BYTE(CLEAN.CLEAN);
    END_IF;
END_IF;

(* revision histroy
hm	18. jun. 2008	rev 1.0
	original release

hm	20. sep. 2008	rev 1.1
	changed length of input string from 20 to 12
*)
(*@KEY@: END_WORKSHEET *)
END_FUNCTION_BLOCK

(* ---- FSTRING_TO_DT.ST ---- *)
(*@PROPERTIES_EX@
TYPE: POU
LOCALE: 0
IEC_LANGUAGE: ST
PLC_TYPE: independent
PROC_TYPE: independent
GROUP: STRINGS
*)
(*@KEY@:DESCRIPTION*)
version 1.0	24. sep. 2008
programmer 	hugo
tested by	oscat

FSTRING_TO_DT converts Formatted String into a DT value.
(*@KEY@:END_DESCRIPTION*)
FUNCTION_BLOCK FSTRING_TO_DT

(*Group:Default*)

VAR_INPUT
	SDT :	oscat_STRING60;
	FMT :	oscat_STRING60;
	IGNORE :	oscat_STRING1 := '*';
	FCHAR :	oscat_STRING1 := '#';
END_VAR

VAR_OUTPUT
	FSTRING_TO_DT :	UDINT;
END_VAR

VAR
	c :	oscat_STRING1;
	tmp :	oscat_STRING20;
	tmp1 :	oscat_STRING1;
	tmp2 :	INT;
	end :	INT;
	dy :	INT;
	dm :	INT;
	dd :	INT;
	th :	INT;
	tm :	INT;
	ts :	INT;
	FSTRING_TO_MONTH :	FSTRING_TO_MONTH;
	IS_NUM :	IS_NUM;
END_VAR

(*@KEY@: WORKSHEET
NAME: FSTRING_TO_DT
IEC_LANGUAGE: ST
*)
dy := 1970;
dm := 1;
dd := 1;
th := 0;
tm := 0;
ts := 0;
FSTRING_TO_DT := UDINT#0;

(* scan input string *)
WHILE (LEN(fmt)>0) DO
	c := LEFT(fmt,1);
	IF EQ_STRING(c,ignore) THEN
		(* skip ignore characters *)
		fmt := DELETE(fmt,1,1);
		IF LEN(sdt)>0 THEN sdt := DELETE(sdt,1,1); END_IF;
	ELSIF EQ_STRING(C,fchar) THEN
		(* format character found skip format char and read identifier *)
		(* store format identifier in c and skip to next char in fmt *)
		IF LEN(fmt) >=2 THEN
		    c := MID(fmt,1,2);
		    fmt := DELETE(fmt,2,1);
        ELSE
		    c := '';
			fmt := '';
		END_IF;
		(* extract the substring until the end of sdt or to next char of fmt *)
		IF LEN(fmt) = 0 THEN
			tmp := sdt;
		ELSE
		    dm := dm;
			(* serach for end of substring *)
            tmp1 := LEFT(fmt,1);
			end := FIND(sdt,tmp1)-1;
            IF end > 0 AND end <= LEN(sdt) THEN
			    tmp := LEFT(sdt, end);
            ELSE
			    tmp := '';
            END_IF;
			sdt := DELETE(sdt, end,1);
        END_IF;

        IS_NUM(str:=tmp);
        IF IS_NUM.IS_NUM THEN
		    tmp2 := STRING_TO_INT(tmp);
        ELSE
		    tmp2 := 0;
	    END_IF;

		(* extract information from substring *)
		IF EQ_STRING(c,'Y') THEN
			dy := tmp2;
			IF dy < 100 THEN dy := dy + 2000; END_IF;
		ELSIF EQ_STRING(c,'M') THEN
			dm := tmp2;
		ELSIF EQ_STRING(c,'N') THEN
		    dm := dm;
            FSTRING_TO_MONTH(MTH:=tmp,LANG:=0);
            dm := FSTRING_TO_MONTH.FSTRING_TO_MONTH;
		ELSIF EQ_STRING(c,'D') THEN
			dd := tmp2;
		ELSIF EQ_STRING(c,'h') THEN
			th := tmp2;
		ELSIF EQ_STRING(c,'m') THEN
			tm := tmp2;
		ELSIF EQ_STRING(c,'s') THEN
			ts := tmp2;
		END_IF;
	ELSE
        tmp1 := LEFT(sdt,1);
	    IF EQ_STRING(c,tmp1) THEN
		    (* skip matching characters *)
		    fmt := DELETE(fmt,1,1);
		    sdt := DELETE(sdt,1,1);
	    ELSE
		    RETURN;
  	    END_IF;
	END_IF;
END_WHILE;

FSTRING_TO_DT := SET_DT(dy,dm,dd,th,tm,ts);

(* revision histroy
hm	24. sep. 2008	rev 1.0
	original release

*)
(*@KEY@: END_WORKSHEET *)
END_FUNCTION_BLOCK

(* ---- FSTRING_TO_DWORD.ST ---- *)
(*@PROPERTIES_EX@
TYPE: POU
LOCALE: 0
IEC_LANGUAGE: ST
PLC_TYPE: independent
PROC_TYPE: independent
GROUP: STRINGS
*)
(*@KEY@:DESCRIPTION*)
version 1.1	20. sep. 2008
programmer 	hugo
tested by		oscat

FSTRING_TO_BYTE converts a formatted string into a byte.
the string can be of the form 2#01010, 8#7234, 16#2AD3 and 1234
(*@KEY@:END_DESCRIPTION*)
FUNCTION_BLOCK FSTRING_TO_DWORD

(*Group:Default*)

VAR_INPUT
	IN :	oscat_STRING40;
END_VAR

VAR_OUTPUT
	FSTRING_TO_DWORD :	DWORD;
END_VAR

VAR
	CLEAN :	CLEAN;
	BIN_TO_DWORD :	BIN_TO_DWORD;
	OCT_TO_DWORD :	OCT_TO_DWORD;
	HEX_TO_DWORD :	HEX_TO_DWORD;
	tmp :	oscat_STRING3;
END_VAR

(*@KEY@: WORKSHEET
NAME: FSTRING_TO_DWORD
IEC_LANGUAGE: ST
*)
tmp := LEFT(IN, 2);
IF EQ_STRING(tmp,'2#') THEN
	(* we need to convert binary *)
    BIN_TO_DWORD(BIN:=RIGHT(in, LEN(in) - 2));
	FSTRING_TO_DWORD := BIN_TO_DWORD.BIN_TO_DWORD;
ELSIF EQ_STRING(tmp,'8#') THEN
	(* weneed to convert octals *)
    OCT_TO_DWORD(OCT:=RIGHT(in, LEN(in) - 2));
	FSTRING_TO_DWORD := OCT_TO_DWORD.OCT_TO_DWORD;
ELSE
    tmp := LEFT(IN, 3);
    IF EQ_STRING(tmp,'16#') THEN
	    (* we need to convert hexadecimal *)
        HEX_TO_DWORD(HEX:=RIGHT(in, LEN(in) - 3));
	    FSTRING_TO_DWORD := HEX_TO_DWORD.HEX_TO_DWORD;
    ELSE
	    (* we assume decimal representation *)
        CLEAN(IN:=in,CX:='0123456789');
	    FSTRING_TO_DWORD := STRING_TO_DWORD(CLEAN.CLEAN);
    END_IF;
END_IF;

(* revision histroy
hm	18. jun. 2008	rev 1.0
	original release

hm	20. sep. 2008	rev 1.1
	changed length of input dtring from 20 to 40

*)
(*@KEY@: END_WORKSHEET *)
END_FUNCTION_BLOCK

(* ---- FSTRING_TO_MONTH.ST ---- *)
(*@PROPERTIES_EX@
TYPE: POU
LOCALE: 0
IEC_LANGUAGE: ST
PLC_TYPE: independent
PROC_TYPE: independent
GROUP: STRINGS
*)
(*@KEY@:DESCRIPTION*)
version 1.2	25. oct 2008
programmer 	hugo
tested by	oscat

FSTRING_TO_MONTH converts a string into a month, the string can be a name for the month or a number.
the function is language sensitve when LANG > 1 and checks for all languages when LANG = 0
(*@KEY@:END_DESCRIPTION*)
FUNCTION_BLOCK FSTRING_TO_MONTH

(*Group:Default*)

VAR_INPUT
	MTH :	oscat_STRING20;
	LANG :	INT;
END_VAR

VAR_OUTPUT
	FSTRING_TO_MONTH :	INT;
END_VAR

VAR
	lx :	INT;
	SETUP_MONTHS :	SETUP_MONTHS;
	MONTHS :	oscat_MONTHS;
	SETUP_MONTHS3 :	SETUP_MONTHS3;
	MONTHS3 :	oscat_MONTHS3;
	SETUP_LANGUAGE :	SETUP_LANGUAGE;
	LANGUAGE :	oscat_LANGUAGE;
	LOWERCASE :	LOWERCASE;
	CAPITALIZE :	CAPITALIZE;
	IS_NUM :	IS_NUM;
END_VAR

(*@KEY@: WORKSHEET
NAME: FSTRING_TO_MONTH
IEC_LANGUAGE: ST
*)
SETUP_MONTHS(MONTHS:=MONTHS);
MONTHS:=SETUP_MONTHS.MONTHS;
SETUP_MONTHS3(MONTHS3:=MONTHS3);
MONTHS3:=SETUP_MONTHS3.MONTHS3;
SETUP_LANGUAGE(LANGUAGE:=LANGUAGE);
LANGUAGE:=SETUP_LANGUAGE.LANGUAGE;

IF LANG = 0 THEN lx := LANGUAGE.DEFAULT; ELSE lx := MIN(LANG, LANGUAGE.LMAX); END_IF;
LOWERCASE(str:=MTH);
CAPITALIZE(str:=LOWERCASE.lowercase);
MTH:=CAPITALIZE.CAPITALIZE;

FOR FSTRING_TO_MONTH := 1 TO 12 DO
	IF EQ_STRING(MTH,MONTHS[lx][FSTRING_TO_MONTH]) THEN RETURN; END_IF;
	IF EQ_STRING(MTH,MONTHS3[lx][FSTRING_TO_MONTH]) THEN RETURN; END_IF;
END_FOR;

(* since no name matched try to decode as integer *)
IS_NUM(str:=MTH);
IF IS_NUM.IS_NUM THEN
	FSTRING_TO_MONTH := STRING_TO_INT(MTH);
ELSE
	FSTRING_TO_MONTH := 0;
END_IF;

(* revision histroy
hm	25. sep. 2008	rev 1.0
	original release

hm	19. oct. 2008	rev 1.1
	changed language setup constants

hm	25. oct. 2008	rev 1.2
	optimized code
*)
(*@KEY@: END_WORKSHEET *)
END_FUNCTION_BLOCK

(* ---- FSTRING_TO_WEEK.ST ---- *)
(*@PROPERTIES_EX@
TYPE: POU
LOCALE: 0
IEC_LANGUAGE: ST
PLC_TYPE: independent
PROC_TYPE: independent
GROUP: STRINGS
*)
(*@KEY@:DESCRIPTION*)
version 1.1	25. oct. 2008
programmer 	hugo
tested by	oscat

FSTRING_TO_WEEK converts a list of weekdays into a byte where each bit represents a day of the week.
bit 6 = mo, 0 = su;
(*@KEY@:END_DESCRIPTION*)
FUNCTION_BLOCK FSTRING_TO_WEEK

(*Group:Default*)

VAR_INPUT
	WEEK :	oscat_STRING60;
	LANG :	INT;
END_VAR

VAR_OUTPUT
	FSTRING_TO_WEEK :	BYTE;
END_VAR

VAR
	pos :	INT;
	FSTRING_TO_WEEKDAY :	FSTRING_TO_WEEKDAY;
END_VAR

(*@KEY@: WORKSHEET
NAME: FSTRING_TO_WEEK
IEC_LANGUAGE: ST
*)
pos := FIND(WEEK, ',');
WHILE pos > 0 DO
    FSTRING_TO_WEEKDAY(WDAY:=MID(WEEK, pos - 1, 1),LANG:=LANG);
	FSTRING_TO_WEEK := FSTRING_TO_WEEK OR SHR_BYTE(BYTE#128, FSTRING_TO_WEEKDAY.FSTRING_TO_WEEKDAY);
	WEEK := RIGHT(WEEK, LEN(Week) - pos);
	pos := FIND(WEEK, ',');
END_WHILE;

FSTRING_TO_WEEKDAY(WDAY:=WEEK,LANG:=LANG);
FSTRING_TO_WEEK := (FSTRING_TO_WEEK OR SHR(BYTE#128, FSTRING_TO_WEEKDAY.FSTRING_TO_WEEKDAY)) AND BYTE#127;

(* revision histroy
hm	18. jun. 2008	rev 1.0
	original release

hm	25. oct. 2008	rev 1.1
	using language defauls and input lang
*)
(*@KEY@: END_WORKSHEET *)
END_FUNCTION_BLOCK

(* ---- FSTRING_TO_WEEKDAY.ST ---- *)
(*@PROPERTIES_EX@
TYPE: POU
LOCALE: 0
IEC_LANGUAGE: ST
PLC_TYPE: independent
PROC_TYPE: independent
GROUP: STRINGS
*)
(*@KEY@:DESCRIPTION*)
version 1.2	25. oct. 2008
programmer 	hugo
tested by	oscat

FSTRING_TO_WEEKDAY converts a weekday string into an integer 1..7.
(*@KEY@:END_DESCRIPTION*)
FUNCTION_BLOCK FSTRING_TO_WEEKDAY

(*Group:Default*)

VAR_INPUT
	WDAY :	oscat_STRING20;
	LANG :	INT;
END_VAR

VAR_OUTPUT
	FSTRING_TO_WEEKDAY :	INT;
END_VAR

VAR
	tmp :	oscat_STRING2;
	i :	INT;
	ly :	INT;
	TRIM :	TRIM;
	SETUP_LANGUAGE :	SETUP_LANGUAGE;
	LANGUAGE :	oscat_LANGUAGE;
	SETUP_WEEKDAYS2 :	SETUP_WEEKDAYS2;
	WEEKDAYS2 :	oscat_WEEKDAYS2;
	LOWERCASE :	LOWERCASE;
	CAPITALIZE :	CAPITALIZE;
	DEC_TO_INT :	DEC_TO_INT;
END_VAR

(*@KEY@: WORKSHEET
NAME: FSTRING_TO_WEEKDAY
IEC_LANGUAGE: ST
*)
SETUP_WEEKDAYS2(WEEKDAYS2:=WEEKDAYS2);
WEEKDAYS2:=SETUP_WEEKDAYS2.WEEKDAYS2;
SETUP_LANGUAGE(LANGUAGE:=LANGUAGE);
LANGUAGE:=SETUP_LANGUAGE.LANGUAGE;

IF LANG = 0 THEN ly := LANGUAGE.DEFAULT; ELSE ly := MIN(LANG, LANGUAGE.LMAX); END_IF;
(* tmp needs to be calculated first otherwise find can return wrong values *)
TRIM(str:=WDAY);
LOWERCASE(str:=TRIM.trim);
tmp:=LOWERCASE.lowercase;
CAPITALIZE(str:=LOWERCASE.lowercase);
tmp:=CAPITALIZE.CAPITALIZE;
FOR i := 1 TO 7 DO
	IF EQ_STRING(WEEKDAYS2[ly][i],tmp) THEN
		FSTRING_TO_WEEKDAY := i;
		RETURN;
	END_IF;
END_FOR;

DEC_TO_INT(DEC:=WDAY);
FSTRING_TO_WEEKDAY:=DEC_TO_INT.DEC_TO_INT;

(* revision histroy
hm	18. jun. 2008	rev 1.0
	original release

hm	18. jul. 2008	rev 1.1
	changed nested call of left(trim()) for compatibility reasons

hm	25. oct. 2008	rev 1.2
	using language constants
*)
(*@KEY@: END_WORKSHEET *)
END_FUNCTION_BLOCK

(* ---- FT_AVG.ST ---- *)
(*@PROPERTIES_EX@
TYPE: POU
LOCALE: 0
IEC_LANGUAGE: ST
PLC_TYPE: independent
PROC_TYPE: independent
GROUP: MATHEMATICAL.FUNCTIONS
*)
(*@KEY@:DESCRIPTION*)
version 1.5	10. mar. 2009
programmer 	hugo
tested by	oscat

this function calculates the moving average over n samples from a sequential input
the input values are shifted into an N deep buffer and the avg of this buffer is diplayed at anytime on the output.
a rst will load the buffer with the current in value..

(*@KEY@:END_DESCRIPTION*)
FUNCTION_BLOCK FT_AVG

(*Group:Default*)

VAR_INPUT
	IN :	REAL;
	E :	BOOL := TRUE;
	N :	INT := INT#32;
	RST :	BOOL;
END_VAR

VAR_OUTPUT
	AVG :	REAL;
END_VAR

VAR
	buff :	delay;
	i :	INT;
	init :	BOOL;
END_VAR

(*@KEY@: WORKSHEET
NAME: FT_AVG
IEC_LANGUAGE: ST
*)
(* limit n to a max of 32 because delay can do max 32 cycles *)
buff.N := LIMIT(0, N, 32);

IF NOT init OR rst THEN
	FOR i := 1 TO N DO
		buff(in := in);
	END_FOR;
	avg := in;
	init := TRUE;
ELSIF E THEN
	buff(in := in);
	avg := avg + (in - buff.out ) / INT_TO_REAL(N);
END_IF;

(* revision history

hm	7. jan. 2007	rev 1.1
	chaged rst logic to load the buffer with the actual input value instead of 0.
	added en input to allow better control of signal flow
	added init to load the buffer with in at startup to avoid rampup at beginning.
	deleted unused variable cnt.

hm	14. jun. 2008	rev 1.2
	set default for input en = TRUE and N = 32

hm	10. oct. 2008	rev 1.3
	improved performance

hm	18. oct. 2008	rev 1.4
	changed input en to e for compatibility reasons

hm	10. mar. 2009	rev 1.5
	added type conversion for compatibility reasons

*)
(*@KEY@: END_WORKSHEET *)
END_FUNCTION_BLOCK

(* ---- FT_DERIV.ST ---- *)
(*@PROPERTIES_EX@
TYPE: POU
LOCALE: 0
IEC_LANGUAGE: ST
PLC_TYPE: independent
PROC_TYPE: independent
GROUP: ENGINEERING.CONTROL
*)
(*@KEY@:DESCRIPTION*)
version 1.5	11. mar. 2009
programmer 	hugo
tested by	oscat

FT_deriv calculates the derivate over the signal "in" with Faktor "K".
a run input enables or stops the calculation, if left unconnected its true and therfore the calculation is executed.
if K is not specified the default is 1.

(*@KEY@:END_DESCRIPTION*)
FUNCTION_BLOCK FT_DERIV

(*Group:Default*)

VAR_INPUT
	IN :	REAL;
	K :	REAL := 1.0;
	RUN :	BOOL := TRUE;
END_VAR

VAR_OUTPUT
	OUT :	REAL;
END_VAR

VAR
	old :	REAL;
	tx :	UDINT;
	last :	UDINT;
	init :	BOOL;
	tc :	REAL;
	T_PLC_US :	T_PLC_US;
END_VAR

(*@KEY@: WORKSHEET
NAME: FT_DERIV
IEC_LANGUAGE: ST
*)
(* read system time *)
T_PLC_US();
tx:= T_PLC_US.T_PLC_US;
tc := UDINT_TO_REAL(tx - last);

(* init on firsat startup *)
IF NOT init THEN
	init := TRUE;
	old := in;
ELSIF run AND tc > 0.0 THEN
	out := (in - old) / tc * 1000000.0 * K;
	old := in;
ELSE
	out := 0.0;
END_IF;

last := tx;

(*
hm 3.1.2007			rev 1.1
	added init code for startup
	set the default for K to 1

hm	15. sep 2007	rev 1.2
	replaced Time() with T_PLC_US for compatibility and performance reasons
	increased accuracy and work in microseconds internally

hm 29 oct 2007	rev 1.3
	prohibit calculation when tx - last = 0 to avoid division by 0 and increase accuracy on fast systems

hm	6. nov. 2008	rev 1.4
	improved performance

hm	11. mar. 2009	rev 1.5
	inproved code
*)

(* read system time *)
T_PLC_US();
tx:= T_PLC_US.T_PLC_US;

(* init on firsat startup *)
IF NOT init THEN
	init := TRUE;
ELSIF run AND tx - last > UDINT#0 THEN
	out := (in - old) / UDINT_TO_REAL(tx - last) * 1000000.0 * K;
ELSE
	out := 0.0;
END_IF;
old := in;
last := tx;

(*
hm 3.1.2007			rev 1.1
	added init code for startup
	set the default for K to 1

hm	15. sep 2007	rev 1.2
	replaced Time() with T_PLC_US for compatibility and performance reasons
	increased accuracy and work in microseconds internally

hm 29 oct 2007	rev 1.3
	prohibit calculation when tx - last = 0 to avoid division by 0 and increase accuracy on fast systems

hm	3. nov. 2008	rev 1.4
	improved performance
*)
(*@KEY@: END_WORKSHEET *)
END_FUNCTION_BLOCK

(* ---- FT_IMP.ST ---- *)
(*@PROPERTIES_EX@
TYPE: POU
LOCALE: 0
IEC_LANGUAGE: ST
PLC_TYPE: independent
PROC_TYPE: independent
GROUP: ENGINEERING.CONTROL
*)
(*@KEY@:DESCRIPTION*)
version 1.1	3 Jan 2007
programmer 	hugo
tested by	tobias

FT_IMP is 	an impulse filter (high pass filter) with the time T and factor K.
(*@KEY@:END_DESCRIPTION*)
FUNCTION_BLOCK FT_IMP

(*Group:Default*)

VAR_INPUT
	IN :	REAL;
	T :	TIME;
	K :	REAL := 1.0;
END_VAR

VAR_OUTPUT
	OUT :	REAL;
END_VAR

VAR
	t1 :	FT_PT1;
END_VAR

(*@KEY@: WORKSHEET
NAME: FT_IMP
IEC_LANGUAGE: ST
*)
T1(in:= in, T:=T);
out := (in - t1.out) * K;

(*
hm 3.1.2007	rev 1.1
	added factor K

*)
(*@KEY@: END_WORKSHEET *)
END_FUNCTION_BLOCK

(* ---- FT_INT.ST ---- *)
(*@PROPERTIES_EX@
TYPE: POU
LOCALE: 0
IEC_LANGUAGE: ST
PLC_TYPE: independent
PROC_TYPE: independent
GROUP: ENGINEERING.CONTROL
*)
(*@KEY@:DESCRIPTION*)
version 2.2	10. mar. 2009
programmer 	hugo
tested by	oscat

FT_int is an integrator with input IN and factor K.
integration is only done while run = true, if run is false integration is stopped and the out remains at the last value.
if run is left unconnected, run is considered true by the function block.
the output ET will display the total integration time from last reset.
the out_min and out_max values can be set to ,imit the output value range.
the default for K is 1.
(*@KEY@:END_DESCRIPTION*)
FUNCTION_BLOCK FT_INT

(*Group:Default*)

VAR_INPUT
	IN :	REAL;
	K :	REAL := 1.0;
	RUN :	BOOL := TRUE;
	RST :	BOOL;
	OUT_MIN :	REAL := REAL#-1.0E-37;
	OUT_MAX :	REAL := REAL#1.0E37;
END_VAR

VAR_OUTPUT
	OUT :	REAL;
	LIM :	BOOL;
END_VAR

VAR
	INTEG :	INTEGRATE;
END_VAR

(*@KEY@: WORKSHEET
NAME: FT_INT
IEC_LANGUAGE: ST
*)
IF rst THEN
	out := 0.0;
ELSE
	integ(X := IN, E := RUN, K := K, Y := out);
	out := integ.Y;
END_IF;

(* limit the outputs *)
IF out >= OUT_MAX THEN
	out := out_max;
	LIM := TRUE;
ELSIF out <= out_min THEN
	out := out_min;
	lim := TRUE;
ELSE
	lim := FALSE;
END_IF;

(*
hm 13.12.2006	rev 1.1
	changed to "trapezregel" which increases accuracy
	before out := out + in * time new: out := out + (in + in_last) / 2 * time

hm 15.1.2007		rev 1.2
	added default for k to be 1.

hm	15.9.2007		rev 1.3
	replaced time() with T_PLC_US for compatibility and performance reason
	increased internal accuracy to microseconds

hm 29. oct 2007		rev 1.4
	changed code so int will not be called is time difference is 0 to increase accuracy on systems
	with cycle times below 1ms

hm	2. dec 2007	 	rev 1.5
	changed code for better performance

hm	5. jan 2008		rev 1.6
	further improvements in performance

hm	8. feb 2008		rev 1.7
	deleted limits +/- 1000 now limit is the range of real
	added variables out1 and out2 to extend the resolution
	corrected an error with elapsed time
	deleted unusfull output ET

hm	13. mar 2008	rev 1.8
	changed preset value out_min to -1e37.
	stop integrator at the limits.

hm	16. mar 2008	rev 1.9
	added type conversion to avoid warning under codesys 3.0

hm	2. jun. 2008	rev 2.0
	rewritten with clear code
	limits can now be set without run

hm	3. nov. 2008	rev 2.1
	optimized code using INTEGRATE and LIMX

hm	10. mar. 2009	rev 2.2
	removed nested comments
*)
(*@KEY@: END_WORKSHEET *)
END_FUNCTION_BLOCK

(* ---- FT_INT2.ST ---- *)
(*@PROPERTIES_EX@
TYPE: POU
LOCALE: 0
IEC_LANGUAGE: ST
PLC_TYPE: independent
PROC_TYPE: independent
GROUP: ENGINEERING.CONTROL
*)
(*@KEY@:DESCRIPTION*)
version 1.2	11. mar. 2009
programmer 	hugo
tested by	oscat

FT_int2 is an integrator with input IN and factor K.
integration is only done while run = true, if run is false integration is stopped and the out remains at the last value.
if run is left unconnected, run is considered true by the function block.
the out_min and out_max values can be set to ,imit the output value range.
the default for K is 1.
FT_INT2 has double presision accuracy (14 digits).
(*@KEY@:END_DESCRIPTION*)
FUNCTION_BLOCK FT_INT2

(*Group:Default*)

VAR_INPUT
	IN :	REAL;
	K :	REAL := 1.0;
	RUN :	BOOL := TRUE;
	RST :	BOOL;
	OUT_MIN :	REAL := REAL#-1.0E-37;
	OUT_MAX :	REAL := REAL#1.0E37;
END_VAR

VAR_OUTPUT
	OUT :	REAL;
	LIM :	BOOL;
END_VAR

VAR
	integ :	INTEGRATE;
	ix :	REAL;
	val :	REAL2;
	R2_ADD :	R2_ADD;
	R2_SET :	R2_SET;
END_VAR

(*@KEY@: WORKSHEET
NAME: FT_INT2
IEC_LANGUAGE: ST
*)
IF RST THEN
	R2_SET(X:=0.0);
	val:=R2_SET.R2_SET;
	out := 0.0;
ELSE
	integ(X := IN, E := RUN, K := K, Y := ix);
	ix := integ.Y;
	R2_ADD(X:=val,Y:=ix);
	val:=R2_ADD.R2_ADD;
	ix := 0.0;
	OUT := val.RX;
END_IF;

(* check output for limits *)
IF out > OUT_MIN AND out < OUT_MAX THEN
	LIM := FALSE;
ELSE
	OUT := LIMIT(OUT_MIN, OUT, OUT_MAX);
	R2_SET(X:=OUT);
	val:=R2_SET.R2_SET;
	LIM := TRUE;
END_IF;

(*	revision history
hm	2. jun. 2008	rev 1.0
	original version

hm	5. nov. 2008	rev 1.1
	rewritten code using integrate

hm	11. mar. 2009	rev 1.2
	real constants updated to new systax using dot

*)
(*@KEY@: END_WORKSHEET *)
END_FUNCTION_BLOCK

(* ---- FT_MIN_MAX.ST ---- *)
(*@PROPERTIES_EX@
TYPE: POU
LOCALE: 0
IEC_LANGUAGE: ST
PLC_TYPE: independent
PROC_TYPE: independent
GROUP: MATHEMATICAL.FUNCTIONS
*)
(*@KEY@:DESCRIPTION*)
version 1.0	1 sep 2006
programmer 	hugo
tested by	tobias

this function block stores the min and max value of an input signal.
when rst is true the mn and mx outputs are set to the in value.
when a rst is never active the function autoresets to the in value at startup.
since the input might not be present at first cycle the mn and mx are set during second cycle.
(*@KEY@:END_DESCRIPTION*)
FUNCTION_BLOCK FT_MIN_MAX

(*Group:Default*)

VAR_INPUT
	IN :	REAL;
	RST :	BOOL;
END_VAR

VAR_OUTPUT
	MX :	REAL;
	MN :	REAL;
END_VAR

VAR
	init :	BOOL;
END_VAR

(*@KEY@: WORKSHEET
NAME: FT_MIN_MAX
IEC_LANGUAGE: ST
*)
IF (rst = TRUE) OR (init = FALSE) THEN
  mn := in;
  mx := in;
  init := TRUE;
ELSIF (in < mn) THEN
  mn := in;
ELSIF (in > mx) THEN
  mx := in;
END_IF;
(*@KEY@: END_WORKSHEET *)
END_FUNCTION_BLOCK

(* ---- FT_PD.ST ---- *)
(*@PROPERTIES_EX@
TYPE: POU
LOCALE: 0
IEC_LANGUAGE: ST
PLC_TYPE: independent
PROC_TYPE: independent
GROUP: ENGINEERING.CONTROL
*)
(*@KEY@:DESCRIPTION*)
version 1.0	3. jun 2008
programmer 	hugo
tested by	tobias

FT_PD is a PD controller.
The PD controller works according to the fomula Y = KP *(IN + DERIV(e) ).
(*@KEY@:END_DESCRIPTION*)
FUNCTION_BLOCK FT_PD

(*Group:Default*)

VAR_INPUT
	IN :	REAL;
	KP :	REAL := 1.0;
	TV :	REAL := 1.0;
END_VAR

VAR_OUTPUT
	Y :	REAL;
END_VAR

VAR
	diff :	FT_DERIV;
END_VAR

(*@KEY@: WORKSHEET
NAME: FT_PD
IEC_LANGUAGE: ST
*)
(* run differentiator *)
diff(IN := IN, K := TV);

(* combine both values *)
Y := KP * (diff.out + IN);

(* revision history
hm 	3. jun. 2008 	rev 1.0
	original version

*)
(*@KEY@: END_WORKSHEET *)
END_FUNCTION_BLOCK

(* ---- FT_PDT1.ST ---- *)
(*@PROPERTIES_EX@
TYPE: POU
LOCALE: 0
IEC_LANGUAGE: ST
PLC_TYPE: independent
PROC_TYPE: independent
GROUP: ENGINEERING.CONTROL
*)
(*@KEY@:DESCRIPTION*)
version 1.0	3. jun 2008
programmer 	hugo
tested by	tobias

FT_PD is a PD controller.
The PD controller works according to the fomula Y = KP *(IN + DERIV(e) ).
(*@KEY@:END_DESCRIPTION*)
FUNCTION_BLOCK FT_PDT1

(*Group:Default*)

VAR_INPUT
	IN :	REAL;
	KP :	REAL := 1.0;
	TV :	REAL := 1.0;
	T1 :	REAL := 1.0;
END_VAR

VAR_OUTPUT
	Y :	REAL;
END_VAR

VAR
	diff :	FT_DERIV;
	TP :	FT_PT1;
END_VAR

(*@KEY@: WORKSHEET
NAME: FT_PDT1
IEC_LANGUAGE: ST
*)
(* run differentiator *)
diff(IN := IN, K := TV);

(* Run PT1 filter *)
tp(in := diff.out, T := REAL_TO_TIME(T1));

(* combine both values *)
Y := KP * (tp.out + IN);

(* revision history
hm 	3. jun. 2008 	rev 1.0
	original version

*)
(*@KEY@: END_WORKSHEET *)
END_FUNCTION_BLOCK

(* ---- FT_PI.ST ---- *)
(*@PROPERTIES_EX@
TYPE: POU
LOCALE: 0
IEC_LANGUAGE: ST
PLC_TYPE: independent
PROC_TYPE: independent
GROUP: ENGINEERING.CONTROL
*)
(*@KEY@:DESCRIPTION*)
version 2.0	3. jun 2008
programmer 	hugo
tested by	tobias

FT_PI is a PI controller.
The PID controller works according to the fomula Y = IN *(KP+ KI * INTEG(e) ).
a rst will reset the integrator to 0
ilim_h and iLim_l set the possible output range of the internal integrator.
the output flags lim will signal that the output limits are active.

default values for KP = 1, KI = 1, ILIM_L = -1E37, iLIM_H = +1E38.
(*@KEY@:END_DESCRIPTION*)
FUNCTION_BLOCK FT_PI

(*Group:Default*)

VAR_INPUT
	IN :	REAL;
	KP :	REAL := 1.0;
	KI :	REAL := 1.0;
	ILIM_L :	REAL := -1.0E38;
	ILIM_H :	REAL := 1.0E38;
	IEN :	BOOL := TRUE;
	RST :	BOOL := FALSE;
END_VAR

VAR_OUTPUT
	Y :	REAL;
	LIM :	BOOL;
END_VAR

VAR
	integ :	FT_INT;
END_VAR

(*@KEY@: WORKSHEET
NAME: FT_PI
IEC_LANGUAGE: ST
*)
(* run integrator *)
integ(IN := IN, K := KI, RUN := IEN, RST := RST, OUT_MIN := ILIM_L, OUT_MAX := ILIM_H);
(* check if integrator has reached its limits and set overflow *)
LIM := integ.LIM;
Y := KP * IN + integ.Out;

(* revision history
hm 	3. jun. 2008 	rev 2.0
	original version

*)
(*@KEY@: END_WORKSHEET *)
END_FUNCTION_BLOCK

(* ---- FT_PID.ST ---- *)
(*@PROPERTIES_EX@
TYPE: POU
LOCALE: 0
IEC_LANGUAGE: ST
PLC_TYPE: independent
PROC_TYPE: independent
GROUP: ENGINEERING.CONTROL
*)
(*@KEY@:DESCRIPTION*)
version 2.1	11. mar. 2009
programmer 	hugo
tested by	tobias

FT_PI is a PI controller.
The PID controller works according to the fomula Y = IN *(KP+ KI * INTEG(e) ).
a rst will reset the integrator to 0
ilim_h and iLim_l set the possible output range of the internal integrator.
the output flags lim will signal that the output limits are active.

default values for KP = 1, KI = 1, ILIM_L = -1E37, iLIM_H = +1E38.
(*@KEY@:END_DESCRIPTION*)
FUNCTION_BLOCK FT_PID

(*Group:Default*)

VAR_INPUT
	IN :	REAL;
	KP :	REAL := 1.0;
	TN :	REAL := 1.0;
	TV :	REAL := 1.0;
	ILIM_L :	REAL := -1.0E38;
	ILIM_H :	REAL := 1.0E38;
	IEN :	BOOL := TRUE;
	RST :	BOOL := FALSE;
END_VAR

VAR_OUTPUT
	Y :	REAL;
	LIM :	BOOL;
END_VAR

VAR
	integ :	FT_INT;
	diff :	FT_DERIV;
END_VAR

(*@KEY@: WORKSHEET
NAME: FT_PID
IEC_LANGUAGE: ST
*)
(* run integrator only if TN > 0 *)
IF TN > 0.0 THEN
	integ(IN := IN, K := 1.0 / TN, RUN := IEN, RST := RST, OUT_MIN := ILIM_L, OUT_MAX := ILIM_H);
ELSE
	integ(RST := FALSE);
END_IF;

(* run differentiator *)
diff(IN := IN, K := TV);

(* combine both values *)
Y := KP * (integ.Out + diff.out + IN);

(* check if integrator has reached its limits and set overflow *)
LIM := integ.LIM;

(* revision history
hm 3. jun. 2008 	rev 2.0
	original version

hm	11. mar. 2009	rev 2.1
	real constants updated to new systax using dot

*)
(*@KEY@: END_WORKSHEET *)
END_FUNCTION_BLOCK
